	VAR jointtarget CDP_3887 := [[1.75, 35.13, 7.04, 0, 47.83, -268.25], [9E9, 9E9, 9E9, 9E9, 9E9, 9E9]];
	VAR jointtarget CDP_3888 := [[0.64, 35.11, 7.08, 0, 47.81, -269.36], [9E9, 9E9, 9E9, 9E9, 9E9, 9E9]];
	VAR jointtarget CDP_3889 := [[-0.47, 35.1, 7.09, 0, 47.81, -270.47], [9E9, 9E9, 9E9, 9E9, 9E9, 9E9]];
	VAR jointtarget CDP_3890 := [[-1.58, 35.13, 7.05, 0, 47.82, -271.58], [9E9, 9E9, 9E9, 9E9, 9E9, 9E9]];
	VAR jointtarget CDP_3891 := [[-2.69, 35.17, 6.97, 0, 47.86, -272.69], [9E9, 9E9, 9E9, 9E9, 9E9, 9E9]];
	VAR jointtarget CDP_3892 := [[-3.8, 35.24, 6.86, 0, 47.9, -273.8], [9E9, 9E9, 9E9, 9E9, 9E9, 9E9]];
	VAR jointtarget CDP_3893 := [[-4.9, 35.33, 6.71, 0, 47.97, -274.9], [9E9, 9E9, 9E9, 9E9, 9E9, 9E9]];
	VAR jointtarget CDP_3894 := [[-6, 35.44, 6.51, 0, 48.05, -276], [9E9, 9E9, 9E9, 9E9, 9E9, 9E9]];
	VAR jointtarget CDP_3895 := [[-7.1, 35.58, 6.28, 0, 48.14, -277.1], [9E9, 9E9, 9E9, 9E9, 9E9, 9E9]];
	VAR jointtarget CDP_3896 := [[-8.19, 35.73, 6.01, 0, 48.25, -278.19], [9E9, 9E9, 9E9, 9E9, 9E9, 9E9]];
	VAR jointtarget CDP_3897 := [[-9.28, 35.92, 5.7, 0, 48.38, -279.28], [9E9, 9E9, 9E9, 9E9, 9E9, 9E9]];
	VAR jointtarget CDP_3898 := [[-10.36, 36.12, 5.35, 0, 48.53, -280.36], [9E9, 9E9, 9E9, 9E9, 9E9, 9E9]];
	VAR jointtarget CDP_3899 := [[-11.43, 36.35, 4.96, 0, 48.69, -281.43], [9E9, 9E9, 9E9, 9E9, 9E9, 9E9]];
	VAR jointtarget CDP_3900 := [[-11.44, 36.35, 4.96, 0, 48.69, -281.78], [9E9, 9E9, 9E9, 9E9, 9E9, 9E9]];
	VAR jointtarget CDP_3901 := [[-11.46, 36.35, 4.95, 0, 48.7, -282.45], [9E9, 9E9, 9E9, 9E9, 9E9, 9E9]];
	VAR jointtarget CDP_3902 := [[-11.48, 36.36, 4.94, 0, 48.7, -283.13], [9E9, 9E9, 9E9, 9E9, 9E9, 9E9]];
	VAR jointtarget CDP_3903 := [[-11.49, 36.36, 4.94, 0, 48.7, -283.81], [9E9, 9E9, 9E9, 9E9, 9E9, 9E9]];
	VAR jointtarget CDP_3904 := [[-11.51, 36.37, 4.93, 0, 48.7, -284.49], [9E9, 9E9, 9E9, 9E9, 9E9, 9E9]];
	VAR jointtarget CDP_3905 := [[-11.53, 36.37, 4.92, 0, 48.71, -285.17], [9E9, 9E9, 9E9, 9E9, 9E9, 9E9]];
	VAR jointtarget CDP_3906 := [[-11.54, 36.38, 4.91, 0, 48.71, -285.84], [9E9, 9E9, 9E9, 9E9, 9E9, 9E9]];
	VAR jointtarget CDP_3907 := [[-11.56, 36.38, 4.9, 0, 48.72, -286.52], [9E9, 9E9, 9E9, 9E9, 9E9, 9E9]];
	VAR jointtarget CDP_3908 := [[-11.57, 36.39, 4.89, 0, 48.72, -287.2], [9E9, 9E9, 9E9, 9E9, 9E9, 9E9]];
	VAR jointtarget CDP_3909 := [[-11.59, 36.39, 4.88, 0, 48.72, -287.88], [9E9, 9E9, 9E9, 9E9, 9E9, 9E9]];
	VAR jointtarget CDP_3910 := [[-11.6, 36.4, 4.87, 0, 48.73, -288.56], [9E9, 9E9, 9E9, 9E9, 9E9, 9E9]];
	VAR jointtarget CDP_3911 := [[-11.62, 36.4, 4.86, 0, 48.73, -289.23], [9E9, 9E9, 9E9, 9E9, 9E9, 9E9]];
	VAR jointtarget CDP_3912 := [[-11.64, 36.41, 4.85, 0, 48.74, -289.91], [9E9, 9E9, 9E9, 9E9, 9E9, 9E9]];
	VAR jointtarget CDP_3913 := [[-11.65, 36.42, 4.84, 0, 48.74, -290.59], [9E9, 9E9, 9E9, 9E9, 9E9, 9E9]];
	VAR jointtarget CDP_3914 := [[-11.67, 36.42, 4.83, 0, 48.75, -291.27], [9E9, 9E9, 9E9, 9E9, 9E9, 9E9]];
	VAR jointtarget CDP_3915 := [[-11.68, 36.43, 4.82, 0, 48.75, -291.94], [9E9, 9E9, 9E9, 9E9, 9E9, 9E9]];
	VAR jointtarget CDP_3916 := [[-11.7, 36.44, 4.81, 0, 48.76, -292.62], [9E9, 9E9, 9E9, 9E9, 9E9, 9E9]];
	VAR jointtarget CDP_3917 := [[-11.71, 36.44, 4.79, 0, 48.76, -293.3], [9E9, 9E9, 9E9, 9E9, 9E9, 9E9]];
	VAR jointtarget CDP_3918 := [[-11.73, 36.45, 4.78, 0, 48.77, -293.98], [9E9, 9E9, 9E9, 9E9, 9E9, 9E9]];
	VAR jointtarget CDP_3919 := [[-11.74, 36.46, 4.77, 0, 48.77, -294.65], [9E9, 9E9, 9E9, 9E9, 9E9, 9E9]];
	VAR jointtarget CDP_3920 := [[-11.8, 36.49, 4.71, 0, 48.79, -295.04], [9E9, 9E9, 9E9, 9E9, 9E9, 9E9]];
	VAR jointtarget CDP_3921 := [[-11.86, 36.52, 4.66, 0, 48.82, -295.11], [9E9, 9E9, 9E9, 9E9, 9E9, 9E9]];
	VAR jointtarget CDP_3922 := [[-11.93, 36.55, 4.61, 0, 48.84, -295.17], [9E9, 9E9, 9E9, 9E9, 9E9, 9E9]];
	VAR jointtarget CDP_3923 := [[-11.99, 36.59, 4.55, 0, 48.86, -295.23], [9E9, 9E9, 9E9, 9E9, 9E9, 9E9]];
	VAR jointtarget CDP_3924 := [[-12.05, 36.62, 4.5, 0, 48.88, -295.29], [9E9, 9E9, 9E9, 9E9, 9E9, 9E9]];
	VAR jointtarget CDP_3925 := [[-12.11, 36.65, 4.44, 0, 48.91, -295.35], [9E9, 9E9, 9E9, 9E9, 9E9, 9E9]];
	VAR jointtarget CDP_3926 := [[-12.17, 36.68, 4.39, 0, 48.93, -295.41], [9E9, 9E9, 9E9, 9E9, 9E9, 9E9]];
	VAR jointtarget CDP_3927 := [[-12.23, 36.71, 4.34, 0, 48.95, -295.47], [9E9, 9E9, 9E9, 9E9, 9E9, 9E9]];
	VAR jointtarget CDP_3928 := [[-12.29, 36.74, 4.28, 0, 48.98, -295.53], [9E9, 9E9, 9E9, 9E9, 9E9, 9E9]];
	VAR jointtarget CDP_3929 := [[-12.35, 36.78, 4.23, 0, 49, -295.59], [9E9, 9E9, 9E9, 9E9, 9E9, 9E9]];
	VAR jointtarget CDP_3930 := [[-12.41, 36.81, 4.17, 0, 49.02, -295.65], [9E9, 9E9, 9E9, 9E9, 9E9, 9E9]];
	VAR jointtarget CDP_3931 := [[-12.47, 36.84, 4.12, 0, 49.04, -295.71], [9E9, 9E9, 9E9, 9E9, 9E9, 9E9]];
	VAR jointtarget CDP_3932 := [[-12.53, 36.87, 4.06, 0, 49.07, -295.77], [9E9, 9E9, 9E9, 9E9, 9E9, 9E9]];
	VAR jointtarget CDP_3933 := [[-12.59, 36.9, 4, 0, 49.09, -295.83], [9E9, 9E9, 9E9, 9E9, 9E9, 9E9]];
	VAR jointtarget CDP_3934 := [[-12.65, 36.94, 3.95, 0, 49.11, -295.89], [9E9, 9E9, 9E9, 9E9, 9E9, 9E9]];
	VAR jointtarget CDP_3935 := [[-12.71, 36.97, 3.89, 0, 49.14, -295.95], [9E9, 9E9, 9E9, 9E9, 9E9, 9E9]];
	VAR jointtarget CDP_3936 := [[-12.77, 37, 3.84, 0, 49.16, -296.01], [9E9, 9E9, 9E9, 9E9, 9E9, 9E9]];
	VAR jointtarget CDP_3937 := [[-12.83, 37.03, 3.78, 0, 49.18, -296.07], [9E9, 9E9, 9E9, 9E9, 9E9, 9E9]];
	VAR jointtarget CDP_3938 := [[-12.89, 37.07, 3.73, 0, 49.21, -296.13], [9E9, 9E9, 9E9, 9E9, 9E9, 9E9]];
	VAR jointtarget CDP_3939 := [[-12.95, 37.1, 3.67, 0, 49.23, -296.19], [9E9, 9E9, 9E9, 9E9, 9E9, 9E9]];
	VAR jointtarget CDP_3940 := [[-13.07, 37.15, 3.58, 0, 49.27, -291.14], [9E9, 9E9, 9E9, 9E9, 9E9, 9E9]];
	VAR jointtarget CDP_3941 := [[-13.19, 37.18, 3.53, 0, 49.29, -280.95], [9E9, 9E9, 9E9, 9E9, 9E9, 9E9]];
	VAR jointtarget CDP_3942 := [[-13.32, 37.18, 3.53, 0, 49.29, -270.75], [9E9, 9E9, 9E9, 9E9, 9E9, 9E9]];
	VAR jointtarget CDP_3943 := [[-13.45, 37.16, 3.57, 0, 49.27, -260.55], [9E9, 9E9, 9E9, 9E9, 9E9, 9E9]];
	VAR jointtarget CDP_3944 := [[-13.57, 37.11, 3.65, 0, 49.24, -250.35], [9E9, 9E9, 9E9, 9E9, 9E9, 9E9]];
	VAR jointtarget CDP_3945 := [[-13.68, 37.04, 3.78, 0, 49.19, -240.14], [9E9, 9E9, 9E9, 9E9, 9E9, 9E9]];
	VAR jointtarget CDP_3946 := [[-13.78, 36.94, 3.94, 0, 49.12, -229.91], [9E9, 9E9, 9E9, 9E9, 9E9, 9E9]];
	VAR jointtarget CDP_3947 := [[-13.86, 36.83, 4.13, 0, 49.04, -219.67], [9E9, 9E9, 9E9, 9E9, 9E9, 9E9]];
	VAR jointtarget CDP_3948 := [[-13.93, 36.71, 4.34, 0, 48.95, -209.41], [9E9, 9E9, 9E9, 9E9, 9E9, 9E9]];
	VAR jointtarget CDP_3949 := [[-13.97, 36.57, 4.58, 0, 48.85, -199.13], [9E9, 9E9, 9E9, 9E9, 9E9, 9E9]];
	VAR jointtarget CDP_3950 := [[-13.99, 36.43, 4.82, 0, 48.75, -188.83], [9E9, 9E9, 9E9, 9E9, 9E9, 9E9]];
	VAR jointtarget CDP_3951 := [[-13.98, 36.29, 5.07, 0, 48.65, -178.5], [9E9, 9E9, 9E9, 9E9, 9E9, 9E9]];
	VAR jointtarget CDP_3952 := [[-13.96, 36.14, 5.31, 0, 48.55, -168.15], [9E9, 9E9, 9E9, 9E9, 9E9, 9E9]];
	VAR jointtarget CDP_3953 := [[-13.91, 36.01, 5.54, 0, 48.45, -157.77], [9E9, 9E9, 9E9, 9E9, 9E9, 9E9]];
	VAR jointtarget CDP_3954 := [[-13.84, 35.89, 5.74, 0, 48.37, -147.38], [9E9, 9E9, 9E9, 9E9, 9E9, 9E9]];
	VAR jointtarget CDP_3955 := [[-13.75, 35.79, 5.92, 0, 48.29, -136.97], [9E9, 9E9, 9E9, 9E9, 9E9, 9E9]];
	VAR jointtarget CDP_3956 := [[-13.64, 35.7, 6.07, 0, 48.23, -126.54], [9E9, 9E9, 9E9, 9E9, 9E9, 9E9]];
	VAR jointtarget CDP_3957 := [[-13.52, 35.64, 6.17, 0, 48.19, -116.09], [9E9, 9E9, 9E9, 9E9, 9E9, 9E9]];
	VAR jointtarget CDP_3958 := [[-13.4, 35.6, 6.24, 0, 48.16, -105.64], [9E9, 9E9, 9E9, 9E9, 9E9, 9E9]];
	VAR jointtarget CDP_3959 := [[-13.27, 35.59, 6.26, 0, 48.15, -95.19], [9E9, 9E9, 9E9, 9E9, 9E9, 9E9]];
	VAR jointtarget CDP_3960 := [[-13.2, 35.59, 6.26, 0, 48.15, -89.96], [9E9, 9E9, 9E9, 9E9, 9E9, 9E9]];
	VAR jointtarget CDP_3961 := [[-13.13, 35.59, 6.26, 0, 48.15, -89.89], [9E9, 9E9, 9E9, 9E9, 9E9, 9E9]];
	VAR jointtarget CDP_3962 := [[-13.06, 35.59, 6.26, 0, 48.15, -89.82], [9E9, 9E9, 9E9, 9E9, 9E9, 9E9]];
	VAR jointtarget CDP_3963 := [[-12.99, 35.59, 6.26, 0, 48.15, -89.75], [9E9, 9E9, 9E9, 9E9, 9E9, 9E9]];
	VAR jointtarget CDP_3964 := [[-12.93, 35.59, 6.26, 0, 48.15, -89.69], [9E9, 9E9, 9E9, 9E9, 9E9, 9E9]];
	VAR jointtarget CDP_3965 := [[-12.86, 35.59, 6.26, 0, 48.16, -89.62], [9E9, 9E9, 9E9, 9E9, 9E9, 9E9]];
	VAR jointtarget CDP_3966 := [[-12.79, 35.59, 6.26, 0, 48.16, -89.55], [9E9, 9E9, 9E9, 9E9, 9E9, 9E9]];
	VAR jointtarget CDP_3967 := [[-12.72, 35.59, 6.26, 0, 48.16, -89.48], [9E9, 9E9, 9E9, 9E9, 9E9, 9E9]];
	VAR jointtarget CDP_3968 := [[-12.65, 35.59, 6.25, 0, 48.16, -89.41], [9E9, 9E9, 9E9, 9E9, 9E9, 9E9]];
	VAR jointtarget CDP_3969 := [[-12.59, 35.59, 6.25, 0, 48.16, -89.35], [9E9, 9E9, 9E9, 9E9, 9E9, 9E9]];
	VAR jointtarget CDP_3970 := [[-12.52, 35.59, 6.25, 0, 48.16, -89.28], [9E9, 9E9, 9E9, 9E9, 9E9, 9E9]];
	VAR jointtarget CDP_3971 := [[-12.45, 35.59, 6.25, 0, 48.16, -89.21], [9E9, 9E9, 9E9, 9E9, 9E9, 9E9]];
	VAR jointtarget CDP_3972 := [[-12.38, 35.59, 6.25, 0, 48.16, -89.14], [9E9, 9E9, 9E9, 9E9, 9E9, 9E9]];
	VAR jointtarget CDP_3973 := [[-12.32, 35.59, 6.25, 0, 48.17, -89.07], [9E9, 9E9, 9E9, 9E9, 9E9, 9E9]];
	VAR jointtarget CDP_3974 := [[-12.25, 35.59, 6.24, 0, 48.17, -89.01], [9E9, 9E9, 9E9, 9E9, 9E9, 9E9]];
	VAR jointtarget CDP_3975 := [[-12.18, 35.59, 6.24, 0, 48.17, -88.94], [9E9, 9E9, 9E9, 9E9, 9E9, 9E9]];
	VAR jointtarget CDP_3976 := [[-12.11, 35.59, 6.24, 0, 48.17, -88.87], [9E9, 9E9, 9E9, 9E9, 9E9, 9E9]];
	VAR jointtarget CDP_3977 := [[-12.04, 35.59, 6.24, 0, 48.17, -88.8], [9E9, 9E9, 9E9, 9E9, 9E9, 9E9]];
	VAR jointtarget CDP_3978 := [[-11.98, 35.59, 6.23, 0, 48.17, -88.74], [9E9, 9E9, 9E9, 9E9, 9E9, 9E9]];
	VAR jointtarget CDP_3979 := [[-11.91, 35.59, 6.23, 0, 48.18, -88.67], [9E9, 9E9, 9E9, 9E9, 9E9, 9E9]];
	VAR jointtarget CDP_3980 := [[-11.89, 35.59, 6.23, 0, 48.18, -88.98], [9E9, 9E9, 9E9, 9E9, 9E9, 9E9]];
	VAR jointtarget CDP_3981 := [[-11.87, 35.59, 6.23, 0, 48.18, -89.63], [9E9, 9E9, 9E9, 9E9, 9E9, 9E9]];
	VAR jointtarget CDP_3982 := [[-11.86, 35.59, 6.23, 0, 48.18, -90.27], [9E9, 9E9, 9E9, 9E9, 9E9, 9E9]];
	VAR jointtarget CDP_3983 := [[-11.84, 35.59, 6.23, 0, 48.18, -90.92], [9E9, 9E9, 9E9, 9E9, 9E9, 9E9]];
	VAR jointtarget CDP_3984 := [[-11.82, 35.59, 6.23, 0, 48.18, -91.56], [9E9, 9E9, 9E9, 9E9, 9E9, 9E9]];
	VAR jointtarget CDP_3985 := [[-11.81, 35.59, 6.23, 0, 48.18, -92.21], [9E9, 9E9, 9E9, 9E9, 9E9, 9E9]];
	VAR jointtarget CDP_3986 := [[-11.79, 35.59, 6.23, 0, 48.18, -92.85], [9E9, 9E9, 9E9, 9E9, 9E9, 9E9]];
	VAR jointtarget CDP_3987 := [[-11.77, 35.59, 6.24, 0, 48.18, -93.5], [9E9, 9E9, 9E9, 9E9, 9E9, 9E9]];
	VAR jointtarget CDP_3988 := [[-11.76, 35.59, 6.24, 0, 48.17, -94.14], [9E9, 9E9, 9E9, 9E9, 9E9, 9E9]];
	VAR jointtarget CDP_3989 := [[-11.74, 35.59, 6.24, 0, 48.17, -94.79], [9E9, 9E9, 9E9, 9E9, 9E9, 9E9]];
	VAR jointtarget CDP_3990 := [[-11.72, 35.58, 6.24, 0, 48.17, -95.43], [9E9, 9E9, 9E9, 9E9, 9E9, 9E9]];
	VAR jointtarget CDP_3991 := [[-11.71, 35.58, 6.25, 0, 48.17, -96.08], [9E9, 9E9, 9E9, 9E9, 9E9, 9E9]];
	VAR jointtarget CDP_3992 := [[-11.69, 35.58, 6.25, 0, 48.17, -96.72], [9E9, 9E9, 9E9, 9E9, 9E9, 9E9]];
	VAR jointtarget CDP_3993 := [[-11.67, 35.58, 6.25, 0, 48.17, -97.37], [9E9, 9E9, 9E9, 9E9, 9E9, 9E9]];
	VAR jointtarget CDP_3994 := [[-11.66, 35.57, 6.26, 0, 48.17, -98.01], [9E9, 9E9, 9E9, 9E9, 9E9, 9E9]];
	VAR jointtarget CDP_3995 := [[-11.64, 35.57, 6.26, 0, 48.16, -98.66], [9E9, 9E9, 9E9, 9E9, 9E9, 9E9]];
	VAR jointtarget CDP_3996 := [[-11.62, 35.57, 6.27, 0, 48.16, -99.31], [9E9, 9E9, 9E9, 9E9, 9E9, 9E9]];
	VAR jointtarget CDP_3997 := [[-11.61, 35.57, 6.27, 0, 48.16, -99.95], [9E9, 9E9, 9E9, 9E9, 9E9, 9E9]];
	VAR jointtarget CDP_3998 := [[-11.59, 35.56, 6.28, 0, 48.16, -100.6], [9E9, 9E9, 9E9, 9E9, 9E9, 9E9]];
	VAR jointtarget CDP_3999 := [[-11.57, 35.56, 6.29, 0, 48.16, -101.24], [9E9, 9E9, 9E9, 9E9, 9E9, 9E9]];
	VAR jointtarget CDP_4000 := [[-10.48, 35.33, 6.68, 0, 47.99, -100.48], [9E9, 9E9, 9E9, 9E9, 9E9, 9E9]];
	VAR jointtarget CDP_4001 := [[-9.38, 35.12, 7.03, 0, 47.85, -99.38], [9E9, 9E9, 9E9, 9E9, 9E9, 9E9]];
	VAR jointtarget CDP_4002 := [[-8.27, 34.94, 7.34, 0, 47.72, -98.27], [9E9, 9E9, 9E9, 9E9, 9E9, 9E9]];
	VAR jointtarget CDP_4003 := [[-7.15, 34.78, 7.61, 0, 47.61, -97.15], [9E9, 9E9, 9E9, 9E9, 9E9, 9E9]];
	VAR jointtarget CDP_4004 := [[-6.03, 34.64, 7.85, 0, 47.51, -96.03], [9E9, 9E9, 9E9, 9E9, 9E9, 9E9]];
	VAR jointtarget CDP_4005 := [[-4.9, 34.53, 8.04, 0, 47.43, -94.9], [9E9, 9E9, 9E9, 9E9, 9E9, 9E9]];
	VAR jointtarget CDP_4006 := [[-3.77, 34.44, 8.19, 0, 47.37, -93.77], [9E9, 9E9, 9E9, 9E9, 9E9, 9E9]];
	VAR jointtarget CDP_4007 := [[-2.64, 34.37, 8.31, 0, 47.32, -92.64], [9E9, 9E9, 9E9, 9E9, 9E9, 9E9]];
	VAR jointtarget CDP_4008 := [[-1.51, 34.33, 8.38, 0, 47.29, -91.51], [9E9, 9E9, 9E9, 9E9, 9E9, 9E9]];
	VAR jointtarget CDP_4009 := [[-0.37, 34.31, 8.41, 0, 47.28, -90.37], [9E9, 9E9, 9E9, 9E9, 9E9, 9E9]];
	VAR jointtarget CDP_4010 := [[0.76, 34.31, 8.41, 0, 47.28, -89.24], [9E9, 9E9, 9E9, 9E9, 9E9, 9E9]];
	VAR jointtarget CDP_4011 := [[1.9, 34.34, 8.36, 0, 47.3, -88.1], [9E9, 9E9, 9E9, 9E9, 9E9, 9E9]];
	VAR jointtarget CDP_4012 := [[3.03, 34.39, 8.27, 0, 47.34, -86.97], [9E9, 9E9, 9E9, 9E9, 9E9, 9E9]];
	VAR jointtarget CDP_4013 := [[4.16, 34.47, 8.14, 0, 47.39, -85.84], [9E9, 9E9, 9E9, 9E9, 9E9, 9E9]];
	VAR jointtarget CDP_4014 := [[5.29, 34.57, 7.98, 0, 47.46, -84.71], [9E9, 9E9, 9E9, 9E9, 9E9, 9E9]];
	VAR jointtarget CDP_4015 := [[6.42, 34.69, 7.77, 0, 47.54, -83.58], [9E9, 9E9, 9E9, 9E9, 9E9, 9E9]];
	VAR jointtarget CDP_4016 := [[7.54, 34.83, 7.52, 0, 47.64, -82.46], [9E9, 9E9, 9E9, 9E9, 9E9, 9E9]];
	VAR jointtarget CDP_4017 := [[8.65, 35, 7.24, 0, 47.76, -81.35], [9E9, 9E9, 9E9, 9E9, 9E9, 9E9]];
	VAR jointtarget CDP_4018 := [[9.76, 35.19, 6.91, 0, 47.9, -80.24], [9E9, 9E9, 9E9, 9E9, 9E9, 9E9]];
	VAR jointtarget CDP_4019 := [[10.86, 35.41, 6.55, 0, 48.05, -79.14], [9E9, 9E9, 9E9, 9E9, 9E9, 9E9]];
	VAR jointtarget CDP_4020 := [[10.87, 35.41, 6.54, 0, 48.05, -79.46], [9E9, 9E9, 9E9, 9E9, 9E9, 9E9]];
	VAR jointtarget CDP_4021 := [[10.89, 35.41, 6.54, 0, 48.05, -80.1], [9E9, 9E9, 9E9, 9E9, 9E9, 9E9]];
	VAR jointtarget CDP_4022 := [[10.91, 35.42, 6.53, 0, 48.05, -80.75], [9E9, 9E9, 9E9, 9E9, 9E9, 9E9]];
	VAR jointtarget CDP_4023 := [[10.92, 35.42, 6.53, 0, 48.06, -81.39], [9E9, 9E9, 9E9, 9E9, 9E9, 9E9]];
	VAR jointtarget CDP_4024 := [[10.94, 35.42, 6.52, 0, 48.06, -82.04], [9E9, 9E9, 9E9, 9E9, 9E9, 9E9]];
	VAR jointtarget CDP_4025 := [[10.96, 35.42, 6.52, 0, 48.06, -82.68], [9E9, 9E9, 9E9, 9E9, 9E9, 9E9]];
	VAR jointtarget CDP_4026 := [[10.97, 35.43, 6.51, 0, 48.06, -83.33], [9E9, 9E9, 9E9, 9E9, 9E9, 9E9]];
	VAR jointtarget CDP_4027 := [[10.99, 35.43, 6.51, 0, 48.06, -83.97], [9E9, 9E9, 9E9, 9E9, 9E9, 9E9]];
	VAR jointtarget CDP_4028 := [[11.01, 35.43, 6.51, 0, 48.06, -84.62], [9E9, 9E9, 9E9, 9E9, 9E9, 9E9]];
	VAR jointtarget CDP_4029 := [[11.02, 35.43, 6.51, 0, 48.06, -85.27], [9E9, 9E9, 9E9, 9E9, 9E9, 9E9]];
	VAR jointtarget CDP_4030 := [[11.04, 35.43, 6.5, 0, 48.07, -85.91], [9E9, 9E9, 9E9, 9E9, 9E9, 9E9]];
	VAR jointtarget CDP_4031 := [[11.06, 35.43, 6.5, 0, 48.07, -86.56], [9E9, 9E9, 9E9, 9E9, 9E9, 9E9]];
	VAR jointtarget CDP_4032 := [[11.07, 35.43, 6.5, 0, 48.07, -87.2], [9E9, 9E9, 9E9, 9E9, 9E9, 9E9]];
	VAR jointtarget CDP_4033 := [[11.09, 35.43, 6.5, 0, 48.07, -87.85], [9E9, 9E9, 9E9, 9E9, 9E9, 9E9]];
	VAR jointtarget CDP_4034 := [[11.11, 35.43, 6.5, 0, 48.07, -88.49], [9E9, 9E9, 9E9, 9E9, 9E9, 9E9]];
	VAR jointtarget CDP_4035 := [[11.13, 35.43, 6.5, 0, 48.07, -89.14], [9E9, 9E9, 9E9, 9E9, 9E9, 9E9]];
	VAR jointtarget CDP_4036 := [[11.14, 35.43, 6.5, 0, 48.07, -89.78], [9E9, 9E9, 9E9, 9E9, 9E9, 9E9]];
	VAR jointtarget CDP_4037 := [[11.16, 35.43, 6.5, 0, 48.07, -90.43], [9E9, 9E9, 9E9, 9E9, 9E9, 9E9]];
	VAR jointtarget CDP_4038 := [[11.18, 35.43, 6.5, 0, 48.07, -91.07], [9E9, 9E9, 9E9, 9E9, 9E9, 9E9]];
	VAR jointtarget CDP_4039 := [[11.19, 35.43, 6.5, 0, 48.07, -91.72], [9E9, 9E9, 9E9, 9E9, 9E9, 9E9]];
	VAR jointtarget CDP_4040 := [[11.26, 35.43, 6.5, 0, 48.07, -91.98], [9E9, 9E9, 9E9, 9E9, 9E9, 9E9]];
	VAR jointtarget CDP_4041 := [[11.33, 35.43, 6.51, 0, 48.06, -91.91], [9E9, 9E9, 9E9, 9E9, 9E9, 9E9]];
	VAR jointtarget CDP_4042 := [[11.4, 35.43, 6.51, 0, 48.06, -91.84], [9E9, 9E9, 9E9, 9E9, 9E9, 9E9]];
	VAR jointtarget CDP_4043 := [[11.47, 35.42, 6.52, 0, 48.06, -91.78], [9E9, 9E9, 9E9, 9E9, 9E9, 9E9]];
	VAR jointtarget CDP_4044 := [[11.53, 35.42, 6.52, 0, 48.06, -91.71], [9E9, 9E9, 9E9, 9E9, 9E9, 9E9]];
	VAR jointtarget CDP_4045 := [[11.6, 35.42, 6.52, 0, 48.06, -91.64], [9E9, 9E9, 9E9, 9E9, 9E9, 9E9]];
	VAR jointtarget CDP_4046 := [[11.67, 35.42, 6.53, 0, 48.06, -91.57], [9E9, 9E9, 9E9, 9E9, 9E9, 9E9]];
	VAR jointtarget CDP_4047 := [[11.74, 35.42, 6.53, 0, 48.05, -91.5], [9E9, 9E9, 9E9, 9E9, 9E9, 9E9]];
	VAR jointtarget CDP_4048 := [[11.81, 35.41, 6.53, 0, 48.05, -91.44], [9E9, 9E9, 9E9, 9E9, 9E9, 9E9]];
	VAR jointtarget CDP_4049 := [[11.87, 35.41, 6.54, 0, 48.05, -91.37], [9E9, 9E9, 9E9, 9E9, 9E9, 9E9]];
	VAR jointtarget CDP_4050 := [[11.94, 35.41, 6.54, 0, 48.05, -91.3], [9E9, 9E9, 9E9, 9E9, 9E9, 9E9]];
	VAR jointtarget CDP_4051 := [[12.01, 35.41, 6.54, 0, 48.05, -91.23], [9E9, 9E9, 9E9, 9E9, 9E9, 9E9]];
	VAR jointtarget CDP_4052 := [[12.08, 35.41, 6.54, 0, 48.05, -91.16], [9E9, 9E9, 9E9, 9E9, 9E9, 9E9]];
	VAR jointtarget CDP_4053 := [[12.15, 35.41, 6.55, 0, 48.05, -91.09], [9E9, 9E9, 9E9, 9E9, 9E9, 9E9]];
	VAR jointtarget CDP_4054 := [[12.21, 35.4, 6.55, 0, 48.05, -91.03], [9E9, 9E9, 9E9, 9E9, 9E9, 9E9]];
	VAR jointtarget CDP_4055 := [[12.28, 35.4, 6.55, 0, 48.05, -90.96], [9E9, 9E9, 9E9, 9E9, 9E9, 9E9]];
	VAR jointtarget CDP_4056 := [[12.35, 35.4, 6.55, 0, 48.04, -90.89], [9E9, 9E9, 9E9, 9E9, 9E9, 9E9]];
	VAR jointtarget CDP_4057 := [[12.42, 35.4, 6.56, 0, 48.04, -90.82], [9E9, 9E9, 9E9, 9E9, 9E9, 9E9]];
	VAR jointtarget CDP_4058 := [[12.49, 35.4, 6.56, 0, 48.04, -90.75], [9E9, 9E9, 9E9, 9E9, 9E9, 9E9]];
	VAR jointtarget CDP_4059 := [[12.55, 35.4, 6.56, 0, 48.04, -90.69], [9E9, 9E9, 9E9, 9E9, 9E9, 9E9]];
	VAR jointtarget CDP_4060 := [[12.69, 35.41, 6.54, 0, 48.05, -85.39], [9E9, 9E9, 9E9, 9E9, 9E9, 9E9]];
	VAR jointtarget CDP_4061 := [[12.81, 35.45, 6.48, 0, 48.08, -74.94], [9E9, 9E9, 9E9, 9E9, 9E9, 9E9]];
	VAR jointtarget CDP_4062 := [[12.93, 35.51, 6.37, 0, 48.12, -64.5], [9E9, 9E9, 9E9, 9E9, 9E9, 9E9]];
	VAR jointtarget CDP_4063 := [[13.04, 35.59, 6.23, 0, 48.18, -54.07], [9E9, 9E9, 9E9, 9E9, 9E9, 9E9]];
	VAR jointtarget CDP_4064 := [[13.13, 35.69, 6.05, 0, 48.25, -43.65], [9E9, 9E9, 9E9, 9E9, 9E9, 9E9]];
	VAR jointtarget CDP_4065 := [[13.2, 35.81, 5.85, 0, 48.34, -33.25], [9E9, 9E9, 9E9, 9E9, 9E9, 9E9]];
	VAR jointtarget CDP_4066 := [[13.25, 35.95, 5.62, 0, 48.43, -22.88], [9E9, 9E9, 9E9, 9E9, 9E9, 9E9]];
	VAR jointtarget CDP_4067 := [[13.28, 36.09, 5.39, 0, 48.53, -12.53], [9E9, 9E9, 9E9, 9E9, 9E9, 9E9]];
	VAR jointtarget CDP_4068 := [[13.29, 36.23, 5.14, 0, 48.63, -2.2], [9E9, 9E9, 9E9, 9E9, 9E9, 9E9]];
	VAR jointtarget CDP_4069 := [[13.27, 36.37, 4.9, 0, 48.73, 8.11], [9E9, 9E9, 9E9, 9E9, 9E9, 9E9]];
	VAR jointtarget CDP_4070 := [[13.23, 36.51, 4.66, 0, 48.83, 18.39], [9E9, 9E9, 9E9, 9E9, 9E9, 9E9]];
	VAR jointtarget CDP_4071 := [[13.17, 36.63, 4.45, 0, 48.92, 28.65], [9E9, 9E9, 9E9, 9E9, 9E9, 9E9]];
	VAR jointtarget CDP_4072 := [[13.08, 36.75, 4.25, 0, 49, 38.9], [9E9, 9E9, 9E9, 9E9, 9E9, 9E9]];
	VAR jointtarget CDP_4073 := [[12.99, 36.84, 4.09, 0, 49.07, 49.12], [9E9, 9E9, 9E9, 9E9, 9E9, 9E9]];
	VAR jointtarget CDP_4074 := [[12.88, 36.91, 3.97, 0, 49.12, 59.33], [9E9, 9E9, 9E9, 9E9, 9E9, 9E9]];
	VAR jointtarget CDP_4075 := [[12.75, 36.96, 3.88, 0, 49.16, 69.54], [9E9, 9E9, 9E9, 9E9, 9E9, 9E9]];
	VAR jointtarget CDP_4076 := [[12.63, 36.99, 3.83, 0, 49.18, 79.73], [9E9, 9E9, 9E9, 9E9, 9E9, 9E9]];
	VAR jointtarget CDP_4077 := [[12.5, 36.99, 3.83, 0, 49.18, 89.93], [9E9, 9E9, 9E9, 9E9, 9E9, 9E9]];
	VAR jointtarget CDP_4078 := [[12.37, 36.96, 3.88, 0, 49.16, 100.13], [9E9, 9E9, 9E9, 9E9, 9E9, 9E9]];
	VAR jointtarget CDP_4079 := [[12.25, 36.91, 3.97, 0, 49.12, 110.33], [9E9, 9E9, 9E9, 9E9, 9E9, 9E9]];
	VAR jointtarget CDP_4080 := [[12.19, 36.88, 4.02, 0, 49.1, 115.43], [9E9, 9E9, 9E9, 9E9, 9E9, 9E9]];
	VAR jointtarget CDP_4081 := [[12.13, 36.85, 4.07, 0, 49.08, 115.37], [9E9, 9E9, 9E9, 9E9, 9E9, 9E9]];
	VAR jointtarget CDP_4082 := [[12.07, 36.82, 4.13, 0, 49.05, 115.31], [9E9, 9E9, 9E9, 9E9, 9E9, 9E9]];
	VAR jointtarget CDP_4083 := [[12.01, 36.79, 4.18, 0, 49.03, 115.25], [9E9, 9E9, 9E9, 9E9, 9E9, 9E9]];
	VAR jointtarget CDP_4084 := [[11.95, 36.75, 4.24, 0, 49.01, 115.19], [9E9, 9E9, 9E9, 9E9, 9E9, 9E9]];
	VAR jointtarget CDP_4085 := [[11.89, 36.72, 4.29, 0, 48.99, 115.13], [9E9, 9E9, 9E9, 9E9, 9E9, 9E9]];
	VAR jointtarget CDP_4086 := [[11.83, 36.69, 4.35, 0, 48.96, 115.07], [9E9, 9E9, 9E9, 9E9, 9E9, 9E9]];
	VAR jointtarget CDP_4087 := [[11.77, 36.66, 4.4, 0, 48.94, 115.01], [9E9, 9E9, 9E9, 9E9, 9E9, 9E9]];
	VAR jointtarget CDP_4088 := [[11.71, 36.63, 4.45, 0, 48.92, 114.95], [9E9, 9E9, 9E9, 9E9, 9E9, 9E9]];
	VAR jointtarget CDP_4089 := [[11.65, 36.6, 4.51, 0, 48.9, 114.89], [9E9, 9E9, 9E9, 9E9, 9E9, 9E9]];
	VAR jointtarget CDP_4090 := [[11.59, 36.57, 4.56, 0, 48.87, 114.83], [9E9, 9E9, 9E9, 9E9, 9E9, 9E9]];
	VAR jointtarget CDP_4091 := [[11.53, 36.54, 4.61, 0, 48.85, 114.77], [9E9, 9E9, 9E9, 9E9, 9E9, 9E9]];
	VAR jointtarget CDP_4092 := [[11.47, 36.5, 4.67, 0, 48.83, 114.71], [9E9, 9E9, 9E9, 9E9, 9E9, 9E9]];
	VAR jointtarget CDP_4093 := [[11.4, 36.47, 4.72, 0, 48.81, 114.64], [9E9, 9E9, 9E9, 9E9, 9E9, 9E9]];
	VAR jointtarget CDP_4094 := [[11.34, 36.44, 4.77, 0, 48.78, 114.58], [9E9, 9E9, 9E9, 9E9, 9E9, 9E9]];
	VAR jointtarget CDP_4095 := [[11.28, 36.41, 4.83, 0, 48.76, 114.52], [9E9, 9E9, 9E9, 9E9, 9E9, 9E9]];
	VAR jointtarget CDP_4096 := [[11.22, 36.38, 4.88, 0, 48.74, 114.46], [9E9, 9E9, 9E9, 9E9, 9E9, 9E9]];
	VAR jointtarget CDP_4097 := [[11.16, 36.35, 4.93, 0, 48.72, 114.4], [9E9, 9E9, 9E9, 9E9, 9E9, 9E9]];
	VAR jointtarget CDP_4098 := [[11.1, 36.32, 4.98, 0, 48.7, 114.34], [9E9, 9E9, 9E9, 9E9, 9E9, 9E9]];
	VAR jointtarget CDP_4099 := [[11.04, 36.29, 5.03, 0, 48.68, 114.28], [9E9, 9E9, 9E9, 9E9, 9E9, 9E9]];
	VAR jointtarget CDP_4100 := [[11.02, 36.28, 5.05, 0, 48.67, 113.93], [9E9, 9E9, 9E9, 9E9, 9E9, 9E9]];
	VAR jointtarget CDP_4101 := [[11.01, 36.28, 5.06, 0, 48.66, 113.26], [9E9, 9E9, 9E9, 9E9, 9E9, 9E9]];
	VAR jointtarget CDP_4102 := [[10.99, 36.27, 5.07, 0, 48.66, 112.58], [9E9, 9E9, 9E9, 9E9, 9E9, 9E9]];
	VAR jointtarget CDP_4103 := [[10.98, 36.26, 5.08, 0, 48.65, 111.9], [9E9, 9E9, 9E9, 9E9, 9E9, 9E9]];
	VAR jointtarget CDP_4104 := [[10.96, 36.26, 5.09, 0, 48.65, 111.22], [9E9, 9E9, 9E9, 9E9, 9E9, 9E9]];
	VAR jointtarget CDP_4105 := [[10.95, 36.25, 5.11, 0, 48.65, 110.55], [9E9, 9E9, 9E9, 9E9, 9E9, 9E9]];
	VAR jointtarget CDP_4106 := [[10.93, 36.24, 5.12, 0, 48.64, 109.87], [9E9, 9E9, 9E9, 9E9, 9E9, 9E9]];
	VAR jointtarget CDP_4107 := [[10.91, 36.24, 5.13, 0, 48.64, 109.19], [9E9, 9E9, 9E9, 9E9, 9E9, 9E9]];
	VAR jointtarget CDP_4108 := [[10.9, 36.23, 5.14, 0, 48.63, 108.51], [9E9, 9E9, 9E9, 9E9, 9E9, 9E9]];
	VAR jointtarget CDP_4109 := [[10.88, 36.23, 5.15, 0, 48.63, 107.83], [9E9, 9E9, 9E9, 9E9, 9E9, 9E9]];
	VAR jointtarget CDP_4110 := [[10.87, 36.22, 5.16, 0, 48.62, 107.16], [9E9, 9E9, 9E9, 9E9, 9E9, 9E9]];
	VAR jointtarget CDP_4111 := [[10.85, 36.21, 5.16, 0, 48.62, 106.48], [9E9, 9E9, 9E9, 9E9, 9E9, 9E9]];
	VAR jointtarget CDP_4112 := [[10.83, 36.21, 5.17, 0, 48.62, 105.8], [9E9, 9E9, 9E9, 9E9, 9E9, 9E9]];
	VAR jointtarget CDP_4113 := [[10.82, 36.2, 5.18, 0, 48.61, 105.12], [9E9, 9E9, 9E9, 9E9, 9E9, 9E9]];
	VAR jointtarget CDP_4114 := [[10.8, 36.2, 5.19, 0, 48.61, 104.44], [9E9, 9E9, 9E9, 9E9, 9E9, 9E9]];
	VAR jointtarget CDP_4115 := [[10.79, 36.2, 5.2, 0, 48.61, 103.77], [9E9, 9E9, 9E9, 9E9, 9E9, 9E9]];
	VAR jointtarget CDP_4116 := [[10.77, 36.19, 5.2, 0, 48.6, 103.09], [9E9, 9E9, 9E9, 9E9, 9E9, 9E9]];
	VAR jointtarget CDP_4117 := [[10.75, 36.19, 5.21, 0, 48.6, 102.41], [9E9, 9E9, 9E9, 9E9, 9E9, 9E9]];
	VAR jointtarget CDP_4118 := [[10.74, 36.18, 5.22, 0, 48.6, 101.73], [9E9, 9E9, 9E9, 9E9, 9E9, 9E9]];
	VAR jointtarget CDP_4119 := [[10.72, 36.18, 5.22, 0, 48.6, 101.05], [9E9, 9E9, 9E9, 9E9, 9E9, 9E9]];
	VAR jointtarget CDP_4120 := [[9.64, 35.97, 5.58, 0, 48.45, 99.64], [9E9, 9E9, 9E9, 9E9, 9E9, 9E9]];
	VAR jointtarget CDP_4121 := [[8.56, 35.78, 5.91, 0, 48.31, 98.56], [9E9, 9E9, 9E9, 9E9, 9E9, 9E9]];
	VAR jointtarget CDP_4122 := [[7.47, 35.61, 6.19, 0, 48.19, 97.47], [9E9, 9E9, 9E9, 9E9, 9E9, 9E9]];
	VAR jointtarget CDP_4123 := [[6.38, 35.47, 6.44, 0, 48.09, 96.38], [9E9, 9E9, 9E9, 9E9, 9E9, 9E9]];
	VAR jointtarget CDP_4124 := [[5.28, 35.35, 6.64, 0, 48.01, 95.28], [9E9, 9E9, 9E9, 9E9, 9E9, 9E9]];
	VAR jointtarget CDP_4125 := [[4.17, 35.25, 6.81, 0, 47.94, 94.17], [9E9, 9E9, 9E9, 9E9, 9E9, 9E9]];
	VAR jointtarget CDP_4126 := [[3.07, 35.18, 6.94, 0, 47.89, 93.07], [9E9, 9E9, 9E9, 9E9, 9E9, 9E9]];
	VAR jointtarget CDP_4127 := [[1.96, 35.13, 7.03, 0, 47.85, 91.96], [9E9, 9E9, 9E9, 9E9, 9E9, 9E9]];
	VAR jointtarget CDP_4128 := [[0.85, 35.1, 7.07, 0, 47.83, 90.85], [9E9, 9E9, 9E9, 9E9, 9E9, 9E9]];
	VAR jointtarget CDP_4129 := [[-0.26, 35.09, 7.09, 0, 47.82, 89.74], [9E9, 9E9, 9E9, 9E9, 9E9, 9E9]];
	VAR jointtarget CDP_4130 := [[-1.37, 35.11, 7.06, 0, 47.84, 88.63], [9E9, 9E9, 9E9, 9E9, 9E9, 9E9]];
	VAR jointtarget CDP_4131 := [[-2.48, 35.15, 6.99, 0, 47.86, 87.52], [9E9, 9E9, 9E9, 9E9, 9E9, 9E9]];
	VAR jointtarget CDP_4132 := [[-3.59, 35.21, 6.88, 0, 47.91, 86.41], [9E9, 9E9, 9E9, 9E9, 9E9, 9E9]];
	VAR jointtarget CDP_4133 := [[-4.7, 35.3, 6.73, 0, 47.97, 85.3], [9E9, 9E9, 9E9, 9E9, 9E9, 9E9]];
	VAR jointtarget CDP_4134 := [[-5.8, 35.4, 6.55, 0, 48.05, 84.2], [9E9, 9E9, 9E9, 9E9, 9E9, 9E9]];
	VAR jointtarget CDP_4135 := [[-6.9, 35.54, 6.32, 0, 48.14, 83.1], [9E9, 9E9, 9E9, 9E9, 9E9, 9E9]];
	VAR jointtarget CDP_4136 := [[-7.99, 35.69, 6.06, 0, 48.25, 82.01], [9E9, 9E9, 9E9, 9E9, 9E9, 9E9]];
	VAR jointtarget CDP_4137 := [[-9.08, 35.87, 5.76, 0, 48.37, 80.92], [9E9, 9E9, 9E9, 9E9, 9E9, 9E9]];
	VAR jointtarget CDP_4138 := [[-10.16, 36.07, 5.42, 0, 48.52, 79.84], [9E9, 9E9, 9E9, 9E9, 9E9, 9E9]];
	VAR jointtarget CDP_4139 := [[-11.23, 36.29, 5.04, 0, 48.67, 78.77], [9E9, 9E9, 9E9, 9E9, 9E9, 9E9]];
	VAR jointtarget CDP_4140 := [[-11.28, 36.3, 5.02, 0, 48.68, 79.81], [9E9, 9E9, 9E9, 9E9, 9E9, 9E9]];
	VAR jointtarget CDP_4141 := [[-11.34, 36.31, 5, 0, 48.69, 81.95], [9E9, 9E9, 9E9, 9E9, 9E9, 9E9]];
	VAR jointtarget CDP_4142 := [[-11.39, 36.31, 4.99, 0, 48.69, 84.09], [9E9, 9E9, 9E9, 9E9, 9E9, 9E9]];
	VAR jointtarget CDP_4143 := [[-11.45, 36.32, 4.99, 0, 48.7, 86.23], [9E9, 9E9, 9E9, 9E9, 9E9, 9E9]];
	VAR jointtarget CDP_4144 := [[-11.5, 36.32, 4.98, 0, 48.7, 88.37], [9E9, 9E9, 9E9, 9E9, 9E9, 9E9]];
	VAR jointtarget CDP_4145 := [[-11.56, 36.32, 4.98, 0, 48.7, 90.51], [9E9, 9E9, 9E9, 9E9, 9E9, 9E9]];
	VAR jointtarget CDP_4146 := [[-11.61, 36.32, 4.99, 0, 48.69, 92.65], [9E9, 9E9, 9E9, 9E9, 9E9, 9E9]];
	VAR jointtarget CDP_4147 := [[-11.67, 36.31, 5, 0, 48.69, 94.78], [9E9, 9E9, 9E9, 9E9, 9E9, 9E9]];
	VAR jointtarget CDP_4148 := [[-11.72, 36.3, 5.01, 0, 48.69, 96.92], [9E9, 9E9, 9E9, 9E9, 9E9, 9E9]];
	VAR jointtarget CDP_4149 := [[-11.78, 36.29, 5.03, 0, 48.68, 99.06], [9E9, 9E9, 9E9, 9E9, 9E9, 9E9]];
	VAR jointtarget CDP_4150 := [[-11.83, 36.28, 5.05, 0, 48.67, 101.2], [9E9, 9E9, 9E9, 9E9, 9E9, 9E9]];
	VAR jointtarget CDP_4151 := [[-11.89, 36.27, 5.07, 0, 48.66, 103.34], [9E9, 9E9, 9E9, 9E9, 9E9, 9E9]];
	VAR jointtarget CDP_4152 := [[-11.94, 36.25, 5.1, 0, 48.65, 105.48], [9E9, 9E9, 9E9, 9E9, 9E9, 9E9]];
	VAR jointtarget CDP_4153 := [[-11.99, 36.23, 5.13, 0, 48.64, 107.63], [9E9, 9E9, 9E9, 9E9, 9E9, 9E9]];
	VAR jointtarget CDP_4154 := [[-12.04, 36.21, 5.17, 0, 48.62, 109.77], [9E9, 9E9, 9E9, 9E9, 9E9, 9E9]];
	VAR jointtarget CDP_4155 := [[-12.09, 36.19, 5.2, 0, 48.6, 111.91], [9E9, 9E9, 9E9, 9E9, 9E9, 9E9]];
	VAR jointtarget CDP_4156 := [[-12.15, 36.17, 5.25, 0, 48.59, 114.05], [9E9, 9E9, 9E9, 9E9, 9E9, 9E9]];
	VAR jointtarget CDP_4157 := [[-12.19, 36.14, 5.29, 0, 48.57, 116.2], [9E9, 9E9, 9E9, 9E9, 9E9, 9E9]];
	VAR jointtarget CDP_4158 := [[-12.24, 36.11, 5.34, 0, 48.55, 118.34], [9E9, 9E9, 9E9, 9E9, 9E9, 9E9]];
	VAR jointtarget CDP_4159 := [[-12.29, 36.08, 5.4, 0, 48.53, 120.49], [9E9, 9E9, 9E9, 9E9, 9E9, 9E9]];
	VAR jointtarget CDP_4160 := [[-12.32, 36.06, 5.43, 0, 48.51, 121.56], [9E9, 9E9, 9E9, 9E9, 9E9, 9E9]];
	VAR jointtarget CDP_4161 := [[-12.35, 36.04, 5.46, 0, 48.5, 121.53], [9E9, 9E9, 9E9, 9E9, 9E9, 9E9]];
	VAR jointtarget CDP_4162 := [[-12.38, 36.02, 5.49, 0, 48.48, 121.5], [9E9, 9E9, 9E9, 9E9, 9E9, 9E9]];
	VAR jointtarget CDP_4163 := [[-12.41, 36, 5.53, 0, 48.47, 121.47], [9E9, 9E9, 9E9, 9E9, 9E9, 9E9]];
	VAR jointtarget CDP_4164 := [[-12.43, 35.98, 5.56, 0, 48.46, 121.44], [9E9, 9E9, 9E9, 9E9, 9E9, 9E9]];
	VAR jointtarget CDP_4165 := [[-12.46, 35.97, 5.59, 0, 48.44, 121.41], [9E9, 9E9, 9E9, 9E9, 9E9, 9E9]];
	VAR jointtarget CDP_4166 := [[-12.49, 35.95, 5.62, 0, 48.43, 121.39], [9E9, 9E9, 9E9, 9E9, 9E9, 9E9]];
	VAR jointtarget CDP_4167 := [[-12.52, 35.93, 5.66, 0, 48.42, 121.36], [9E9, 9E9, 9E9, 9E9, 9E9, 9E9]];
	VAR jointtarget CDP_4168 := [[-12.55, 35.91, 5.69, 0, 48.4, 121.33], [9E9, 9E9, 9E9, 9E9, 9E9, 9E9]];
	VAR jointtarget CDP_4169 := [[-12.58, 35.89, 5.72, 0, 48.39, 121.3], [9E9, 9E9, 9E9, 9E9, 9E9, 9E9]];
	VAR jointtarget CDP_4170 := [[-12.61, 35.87, 5.75, 0, 48.38, 121.27], [9E9, 9E9, 9E9, 9E9, 9E9, 9E9]];
	VAR jointtarget CDP_4171 := [[-12.63, 35.85, 5.79, 0, 48.36, 121.24], [9E9, 9E9, 9E9, 9E9, 9E9, 9E9]];
	VAR jointtarget CDP_4172 := [[-12.66, 35.83, 5.82, 0, 48.35, 121.21], [9E9, 9E9, 9E9, 9E9, 9E9, 9E9]];
	VAR jointtarget CDP_4173 := [[-12.69, 35.81, 5.85, 0, 48.34, 121.18], [9E9, 9E9, 9E9, 9E9, 9E9, 9E9]];
	VAR jointtarget CDP_4174 := [[-12.72, 35.79, 5.88, 0, 48.32, 121.16], [9E9, 9E9, 9E9, 9E9, 9E9, 9E9]];
	VAR jointtarget CDP_4175 := [[-12.75, 35.78, 5.92, 0, 48.31, 121.13], [9E9, 9E9, 9E9, 9E9, 9E9, 9E9]];
	VAR jointtarget CDP_4176 := [[-12.78, 35.76, 5.95, 0, 48.3, 121.1], [9E9, 9E9, 9E9, 9E9, 9E9, 9E9]];
	VAR jointtarget CDP_4177 := [[-12.81, 35.74, 5.98, 0, 48.28, 121.07], [9E9, 9E9, 9E9, 9E9, 9E9, 9E9]];
	VAR jointtarget CDP_4178 := [[-12.84, 35.72, 6.01, 0, 48.27, 121.04], [9E9, 9E9, 9E9, 9E9, 9E9, 9E9]];
	VAR jointtarget CDP_4179 := [[-12.86, 35.7, 6.04, 0, 48.26, 121.01], [9E9, 9E9, 9E9, 9E9, 9E9, 9E9]];
	VAR jointtarget CDP_4180 := [[-13.02, 35.63, 6.17, 0, 48.2, 114.17], [9E9, 9E9, 9E9, 9E9, 9E9, 9E9]];
	VAR jointtarget CDP_4181 := [[-13.18, 35.59, 6.23, 0, 48.18, 100.62], [9E9, 9E9, 9E9, 9E9, 9E9, 9E9]];
	VAR jointtarget CDP_4182 := [[-13.34, 35.6, 6.21, 0, 48.19, 87.07], [9E9, 9E9, 9E9, 9E9, 9E9, 9E9]];
	VAR jointtarget CDP_4183 := [[-13.5, 35.65, 6.12, 0, 48.22, 73.52], [9E9, 9E9, 9E9, 9E9, 9E9, 9E9]];
	VAR jointtarget CDP_4184 := [[-13.64, 35.74, 5.97, 0, 48.29, 59.99], [9E9, 9E9, 9E9, 9E9, 9E9, 9E9]];
	VAR jointtarget CDP_4185 := [[-13.76, 35.87, 5.76, 0, 48.37, 46.48], [9E9, 9E9, 9E9, 9E9, 9E9, 9E9]];
	VAR jointtarget CDP_4186 := [[-13.85, 36.01, 5.51, 0, 48.48, 33.01], [9E9, 9E9, 9E9, 9E9, 9E9, 9E9]];
	VAR jointtarget CDP_4187 := [[-13.91, 36.18, 5.22, 0, 48.6, 19.56], [9E9, 9E9, 9E9, 9E9, 9E9, 9E9]];
	VAR jointtarget CDP_4188 := [[-13.92, 36.36, 4.91, 0, 48.73, 6.16], [9E9, 9E9, 9E9, 9E9, 9E9, 9E9]];
	VAR jointtarget CDP_4189 := [[-13.9, 36.54, 4.61, 0, 48.85, -7.21], [9E9, 9E9, 9E9, 9E9, 9E9, 9E9]];
	VAR jointtarget CDP_4190 := [[-13.85, 36.71, 4.32, 0, 48.97, -20.54], [9E9, 9E9, 9E9, 9E9, 9E9, 9E9]];
	VAR jointtarget CDP_4191 := [[-13.76, 36.86, 4.06, 0, 49.08, -33.84], [9E9, 9E9, 9E9, 9E9, 9E9, 9E9]];
	VAR jointtarget CDP_4192 := [[-13.64, 36.98, 3.85, 0, 49.17, -47.11], [9E9, 9E9, 9E9, 9E9, 9E9, 9E9]];
	VAR jointtarget CDP_4193 := [[-13.5, 37.07, 3.7, 0, 49.23, -60.35], [9E9, 9E9, 9E9, 9E9, 9E9, 9E9]];
	VAR jointtarget CDP_4194 := [[-13.34, 37.12, 3.61, 0, 49.27, -73.59], [9E9, 9E9, 9E9, 9E9, 9E9, 9E9]];
	VAR jointtarget CDP_4195 := [[-13.18, 37.13, 3.59, 0, 49.28, -86.81], [9E9, 9E9, 9E9, 9E9, 9E9, 9E9]];
	VAR jointtarget CDP_4196 := [[-13.02, 37.1, 3.65, 0, 49.26, -100.04], [9E9, 9E9, 9E9, 9E9, 9E9, 9E9]];
	VAR jointtarget CDP_4197 := [[-12.88, 37.03, 3.77, 0, 49.2, -113.28], [9E9, 9E9, 9E9, 9E9, 9E9, 9E9]];
	VAR jointtarget CDP_4198 := [[-12.75, 36.92, 3.96, 0, 49.13, -126.54], [9E9, 9E9, 9E9, 9E9, 9E9, 9E9]];
	VAR jointtarget CDP_4199 := [[-12.64, 36.78, 4.19, 0, 49.03, -139.82], [9E9, 9E9, 9E9, 9E9, 9E9, 9E9]];
	VAR jointtarget CDP_4200 := [[-12.62, 36.74, 4.26, 0, 49, -146.49], [9E9, 9E9, 9E9, 9E9, 9E9, 9E9]];
	VAR jointtarget CDP_4201 := [[-12.59, 36.7, 4.33, 0, 48.97, -146.47], [9E9, 9E9, 9E9, 9E9, 9E9, 9E9]];
	VAR jointtarget CDP_4202 := [[-12.57, 36.66, 4.4, 0, 48.94, -146.44], [9E9, 9E9, 9E9, 9E9, 9E9, 9E9]];
	VAR jointtarget CDP_4203 := [[-12.54, 36.62, 4.48, 0, 48.91, -146.42], [9E9, 9E9, 9E9, 9E9, 9E9, 9E9]];
	VAR jointtarget CDP_4204 := [[-12.52, 36.57, 4.55, 0, 48.88, -146.4], [9E9, 9E9, 9E9, 9E9, 9E9, 9E9]];
	VAR jointtarget CDP_4205 := [[-12.49, 36.53, 4.62, 0, 48.85, -146.37], [9E9, 9E9, 9E9, 9E9, 9E9, 9E9]];
	VAR jointtarget CDP_4206 := [[-12.47, 36.49, 4.69, 0, 48.82, -146.35], [9E9, 9E9, 9E9, 9E9, 9E9, 9E9]];
	VAR jointtarget CDP_4207 := [[-12.44, 36.45, 4.76, 0, 48.79, -146.32], [9E9, 9E9, 9E9, 9E9, 9E9, 9E9]];
	VAR jointtarget CDP_4208 := [[-12.42, 36.41, 4.83, 0, 48.76, -146.3], [9E9, 9E9, 9E9, 9E9, 9E9, 9E9]];
	VAR jointtarget CDP_4209 := [[-12.39, 36.37, 4.9, 0, 48.73, -146.27], [9E9, 9E9, 9E9, 9E9, 9E9, 9E9]];
	VAR jointtarget CDP_4210 := [[-12.37, 36.33, 4.97, 0, 48.7, -146.25], [9E9, 9E9, 9E9, 9E9, 9E9, 9E9]];
	VAR jointtarget CDP_4211 := [[-12.34, 36.29, 5.04, 0, 48.67, -146.22], [9E9, 9E9, 9E9, 9E9, 9E9, 9E9]];
	VAR jointtarget CDP_4212 := [[-12.32, 36.25, 5.11, 0, 48.64, -146.2], [9E9, 9E9, 9E9, 9E9, 9E9, 9E9]];
	VAR jointtarget CDP_4213 := [[-12.29, 36.2, 5.18, 0, 48.61, -146.17], [9E9, 9E9, 9E9, 9E9, 9E9, 9E9]];
	VAR jointtarget CDP_4214 := [[-12.27, 36.16, 5.25, 0, 48.58, -146.15], [9E9, 9E9, 9E9, 9E9, 9E9, 9E9]];
	VAR jointtarget CDP_4215 := [[-12.24, 36.12, 5.32, 0, 48.56, -146.12], [9E9, 9E9, 9E9, 9E9, 9E9, 9E9]];
	VAR jointtarget CDP_4216 := [[-12.22, 36.08, 5.39, 0, 48.53, -146.1], [9E9, 9E9, 9E9, 9E9, 9E9, 9E9]];
	VAR jointtarget CDP_4217 := [[-12.19, 36.04, 5.46, 0, 48.5, -146.07], [9E9, 9E9, 9E9, 9E9, 9E9, 9E9]];
	VAR jointtarget CDP_4218 := [[-12.17, 36, 5.53, 0, 48.47, -146.05], [9E9, 9E9, 9E9, 9E9, 9E9, 9E9]];
	VAR jointtarget CDP_4219 := [[-12.14, 35.96, 5.6, 0, 48.44, -146.02], [9E9, 9E9, 9E9, 9E9, 9E9, 9E9]];
	VAR jointtarget CDP_4220 := [[-12.14, 35.95, 5.62, 0, 48.43, -145.46], [9E9, 9E9, 9E9, 9E9, 9E9, 9E9]];
	VAR jointtarget CDP_4221 := [[-12.13, 35.93, 5.64, 0, 48.42, -144.35], [9E9, 9E9, 9E9, 9E9, 9E9, 9E9]];
	VAR jointtarget CDP_4222 := [[-12.12, 35.92, 5.66, 0, 48.41, -143.24], [9E9, 9E9, 9E9, 9E9, 9E9, 9E9]];
	VAR jointtarget CDP_4223 := [[-12.11, 35.91, 5.69, 0, 48.4, -142.13], [9E9, 9E9, 9E9, 9E9, 9E9, 9E9]];
	VAR jointtarget CDP_4224 := [[-12.1, 35.9, 5.71, 0, 48.4, -141.01], [9E9, 9E9, 9E9, 9E9, 9E9, 9E9]];
	VAR jointtarget CDP_4225 := [[-12.09, 35.89, 5.73, 0, 48.39, -139.9], [9E9, 9E9, 9E9, 9E9, 9E9, 9E9]];
	VAR jointtarget CDP_4226 := [[-12.08, 35.87, 5.75, 0, 48.38, -138.79], [9E9, 9E9, 9E9, 9E9, 9E9, 9E9]];
	VAR jointtarget CDP_4227 := [[-12.07, 35.86, 5.76, 0, 48.37, -137.68], [9E9, 9E9, 9E9, 9E9, 9E9, 9E9]];
	VAR jointtarget CDP_4228 := [[-12.06, 35.85, 5.78, 0, 48.36, -136.56], [9E9, 9E9, 9E9, 9E9, 9E9, 9E9]];
	VAR jointtarget CDP_4229 := [[-12.05, 35.84, 5.8, 0, 48.36, -135.45], [9E9, 9E9, 9E9, 9E9, 9E9, 9E9]];
	VAR jointtarget CDP_4230 := [[-12.04, 35.83, 5.82, 0, 48.35, -134.34], [9E9, 9E9, 9E9, 9E9, 9E9, 9E9]];
	VAR jointtarget CDP_4231 := [[-12.03, 35.82, 5.84, 0, 48.34, -133.22], [9E9, 9E9, 9E9, 9E9, 9E9, 9E9]];
	VAR jointtarget CDP_4232 := [[-12.02, 35.81, 5.86, 0, 48.34, -132.11], [9E9, 9E9, 9E9, 9E9, 9E9, 9E9]];
	VAR jointtarget CDP_4233 := [[-12.01, 35.8, 5.87, 0, 48.33, -130.99], [9E9, 9E9, 9E9, 9E9, 9E9, 9E9]];
	VAR jointtarget CDP_4234 := [[-12, 35.79, 5.89, 0, 48.32, -129.88], [9E9, 9E9, 9E9, 9E9, 9E9, 9E9]];
	VAR jointtarget CDP_4235 := [[-11.99, 35.78, 5.91, 0, 48.32, -128.76], [9E9, 9E9, 9E9, 9E9, 9E9, 9E9]];
	VAR jointtarget CDP_4236 := [[-11.98, 35.77, 5.92, 0, 48.31, -127.65], [9E9, 9E9, 9E9, 9E9, 9E9, 9E9]];
	VAR jointtarget CDP_4237 := [[-11.97, 35.76, 5.94, 0, 48.3, -126.53], [9E9, 9E9, 9E9, 9E9, 9E9, 9E9]];
	VAR jointtarget CDP_4238 := [[-11.96, 35.75, 5.95, 0, 48.3, -125.42], [9E9, 9E9, 9E9, 9E9, 9E9, 9E9]];
	VAR jointtarget CDP_4239 := [[-11.95, 35.74, 5.97, 0, 48.29, -124.3], [9E9, 9E9, 9E9, 9E9, 9E9, 9E9]];
	VAR jointtarget CDP_4240 := [[-11.94, 35.73, 5.98, 0, 48.29, -123.74], [9E9, 9E9, 9E9, 9E9, 9E9, 9E9]];
	VAR jointtarget CDP_4241 := [[-11.93, 35.72, 5.99, 0, 48.28, -123.73], [9E9, 9E9, 9E9, 9E9, 9E9, 9E9]];
	VAR jointtarget CDP_4242 := [[-11.92, 35.72, 6, 0, 48.28, -123.72], [9E9, 9E9, 9E9, 9E9, 9E9, 9E9]];
	VAR jointtarget CDP_4243 := [[-11.9, 35.71, 6.02, 0, 48.27, -123.71], [9E9, 9E9, 9E9, 9E9, 9E9, 9E9]];
	VAR jointtarget CDP_4244 := [[-11.89, 35.7, 6.03, 0, 48.27, -123.7], [9E9, 9E9, 9E9, 9E9, 9E9, 9E9]];
	VAR jointtarget CDP_4245 := [[-11.88, 35.69, 6.04, 0, 48.26, -123.69], [9E9, 9E9, 9E9, 9E9, 9E9, 9E9]];
	VAR jointtarget CDP_4246 := [[-11.87, 35.69, 6.06, 0, 48.26, -123.68], [9E9, 9E9, 9E9, 9E9, 9E9, 9E9]];
	VAR jointtarget CDP_4247 := [[-11.86, 35.68, 6.07, 0, 48.25, -123.66], [9E9, 9E9, 9E9, 9E9, 9E9, 9E9]];
	VAR jointtarget CDP_4248 := [[-11.85, 35.67, 6.08, 0, 48.25, -123.65], [9E9, 9E9, 9E9, 9E9, 9E9, 9E9]];
	VAR jointtarget CDP_4249 := [[-11.84, 35.66, 6.09, 0, 48.24, -123.64], [9E9, 9E9, 9E9, 9E9, 9E9, 9E9]];
	VAR jointtarget CDP_4250 := [[-11.83, 35.65, 6.11, 0, 48.24, -123.63], [9E9, 9E9, 9E9, 9E9, 9E9, 9E9]];
	VAR jointtarget CDP_4251 := [[-11.82, 35.65, 6.12, 0, 48.24, -123.62], [9E9, 9E9, 9E9, 9E9, 9E9, 9E9]];
	VAR jointtarget CDP_4252 := [[-11.81, 35.64, 6.13, 0, 48.23, -123.61], [9E9, 9E9, 9E9, 9E9, 9E9, 9E9]];
	VAR jointtarget CDP_4253 := [[-11.8, 35.63, 6.14, 0, 48.23, -123.6], [9E9, 9E9, 9E9, 9E9, 9E9, 9E9]];
	VAR jointtarget CDP_4254 := [[-11.79, 35.62, 6.16, 0, 48.22, -123.59], [9E9, 9E9, 9E9, 9E9, 9E9, 9E9]];
	VAR jointtarget CDP_4255 := [[-11.78, 35.61, 6.17, 0, 48.22, -123.58], [9E9, 9E9, 9E9, 9E9, 9E9, 9E9]];
	VAR jointtarget CDP_4256 := [[-11.77, 35.61, 6.18, 0, 48.21, -123.57], [9E9, 9E9, 9E9, 9E9, 9E9, 9E9]];
	VAR jointtarget CDP_4257 := [[-11.76, 35.6, 6.19, 0, 48.21, -123.56], [9E9, 9E9, 9E9, 9E9, 9E9, 9E9]];
	VAR jointtarget CDP_4258 := [[-11.75, 35.59, 6.21, 0, 48.2, -123.55], [9E9, 9E9, 9E9, 9E9, 9E9, 9E9]];
	VAR jointtarget CDP_4259 := [[-11.74, 35.58, 6.22, 0, 48.2, -123.54], [9E9, 9E9, 9E9, 9E9, 9E9, 9E9]];
	VAR jointtarget CDP_4260 := [[-10.65, 35.35, 6.62, 0, 48.03, -100.65], [9E9, 9E9, 9E9, 9E9, 9E9, 9E9]];
	VAR jointtarget CDP_4261 := [[-9.55, 35.14, 6.97, 0, 47.88, -99.55], [9E9, 9E9, 9E9, 9E9, 9E9, 9E9]];
	VAR jointtarget CDP_4262 := [[-8.44, 34.95, 7.29, 0, 47.75, -98.44], [9E9, 9E9, 9E9, 9E9, 9E9, 9E9]];
	VAR jointtarget CDP_4263 := [[-7.33, 34.79, 7.57, 0, 47.64, -97.33], [9E9, 9E9, 9E9, 9E9, 9E9, 9E9]];
	VAR jointtarget CDP_4264 := [[-6.21, 34.65, 7.81, 0, 47.54, -96.21], [9E9, 9E9, 9E9, 9E9, 9E9, 9E9]];
	VAR jointtarget CDP_4265 := [[-5.09, 34.53, 8.01, 0, 47.46, -95.09], [9E9, 9E9, 9E9, 9E9, 9E9, 9E9]];
	VAR jointtarget CDP_4266 := [[-3.96, 34.44, 8.17, 0, 47.39, -93.96], [9E9, 9E9, 9E9, 9E9, 9E9, 9E9]];
	VAR jointtarget CDP_4267 := [[-2.83, 34.37, 8.29, 0, 47.34, -92.83], [9E9, 9E9, 9E9, 9E9, 9E9, 9E9]];
	VAR jointtarget CDP_4268 := [[-1.7, 34.32, 8.37, 0, 47.31, -91.7], [9E9, 9E9, 9E9, 9E9, 9E9, 9E9]];
	VAR jointtarget CDP_4269 := [[-0.56, 34.3, 8.41, 0, 47.3, -90.56], [9E9, 9E9, 9E9, 9E9, 9E9, 9E9]];
	VAR jointtarget CDP_4270 := [[0.57, 34.3, 8.41, 0, 47.3, -89.43], [9E9, 9E9, 9E9, 9E9, 9E9, 9E9]];
	VAR jointtarget CDP_4271 := [[1.7, 34.32, 8.37, 0, 47.31, -88.3], [9E9, 9E9, 9E9, 9E9, 9E9, 9E9]];
	VAR jointtarget CDP_4272 := [[2.84, 34.37, 8.29, 0, 47.35, -87.16], [9E9, 9E9, 9E9, 9E9, 9E9, 9E9]];
	VAR jointtarget CDP_4273 := [[3.97, 34.44, 8.17, 0, 47.39, -86.03], [9E9, 9E9, 9E9, 9E9, 9E9, 9E9]];
	VAR jointtarget CDP_4274 := [[5.09, 34.53, 8.01, 0, 47.46, -84.91], [9E9, 9E9, 9E9, 9E9, 9E9, 9E9]];
	VAR jointtarget CDP_4275 := [[6.22, 34.65, 7.81, 0, 47.54, -83.78], [9E9, 9E9, 9E9, 9E9, 9E9, 9E9]];
	VAR jointtarget CDP_4276 := [[7.34, 34.79, 7.57, 0, 47.64, -82.66], [9E9, 9E9, 9E9, 9E9, 9E9, 9E9]];
	VAR jointtarget CDP_4277 := [[8.45, 34.95, 7.29, 0, 47.75, -81.55], [9E9, 9E9, 9E9, 9E9, 9E9, 9E9]];
	VAR jointtarget CDP_4278 := [[9.56, 35.14, 6.97, 0, 47.89, -80.44], [9E9, 9E9, 9E9, 9E9, 9E9, 9E9]];
	VAR jointtarget CDP_4279 := [[10.65, 35.35, 6.61, 0, 48.03, -79.35], [9E9, 9E9, 9E9, 9E9, 9E9, 9E9]];
	VAR jointtarget CDP_4280 := [[10.71, 35.36, 6.59, 0, 48.04, -78.19], [9E9, 9E9, 9E9, 9E9, 9E9, 9E9]];
	VAR jointtarget CDP_4281 := [[10.76, 35.38, 6.57, 0, 48.05, -75.95], [9E9, 9E9, 9E9, 9E9, 9E9, 9E9]];
	VAR jointtarget CDP_4282 := [[10.82, 35.4, 6.54, 0, 48.06, -73.7], [9E9, 9E9, 9E9, 9E9, 9E9, 9E9]];
	VAR jointtarget CDP_4283 := [[10.87, 35.41, 6.51, 0, 48.08, -71.45], [9E9, 9E9, 9E9, 9E9, 9E9, 9E9]];
	VAR jointtarget CDP_4284 := [[10.92, 35.44, 6.47, 0, 48.09, -69.2], [9E9, 9E9, 9E9, 9E9, 9E9, 9E9]];
	VAR jointtarget CDP_4285 := [[10.97, 35.46, 6.43, 0, 48.11, -66.96], [9E9, 9E9, 9E9, 9E9, 9E9, 9E9]];
	VAR jointtarget CDP_4286 := [[11.03, 35.49, 6.39, 0, 48.13, -64.72], [9E9, 9E9, 9E9, 9E9, 9E9, 9E9]];
	VAR jointtarget CDP_4287 := [[11.07, 35.51, 6.34, 0, 48.15, -62.47], [9E9, 9E9, 9E9, 9E9, 9E9, 9E9]];
	VAR jointtarget CDP_4288 := [[11.12, 35.54, 6.29, 0, 48.17, -60.23], [9E9, 9E9, 9E9, 9E9, 9E9, 9E9]];
	VAR jointtarget CDP_4289 := [[11.17, 35.57, 6.23, 0, 48.19, -57.99], [9E9, 9E9, 9E9, 9E9, 9E9, 9E9]];
	VAR jointtarget CDP_4290 := [[11.22, 35.61, 6.18, 0, 48.22, -55.75], [9E9, 9E9, 9E9, 9E9, 9E9, 9E9]];
	VAR jointtarget CDP_4291 := [[11.26, 35.64, 6.11, 0, 48.24, -53.51], [9E9, 9E9, 9E9, 9E9, 9E9, 9E9]];
	VAR jointtarget CDP_4292 := [[11.3, 35.68, 6.05, 0, 48.27, -51.27], [9E9, 9E9, 9E9, 9E9, 9E9, 9E9]];
	VAR jointtarget CDP_4293 := [[11.35, 35.72, 5.98, 0, 48.3, -49.04], [9E9, 9E9, 9E9, 9E9, 9E9, 9E9]];
	VAR jointtarget CDP_4294 := [[11.39, 35.76, 5.91, 0, 48.32, -46.8], [9E9, 9E9, 9E9, 9E9, 9E9, 9E9]];
	VAR jointtarget CDP_4295 := [[11.43, 35.81, 5.84, 0, 48.36, -44.57], [9E9, 9E9, 9E9, 9E9, 9E9, 9E9]];
	VAR jointtarget CDP_4296 := [[11.46, 35.85, 5.76, 0, 48.39, -42.34], [9E9, 9E9, 9E9, 9E9, 9E9, 9E9]];
	VAR jointtarget CDP_4297 := [[11.5, 35.9, 5.68, 0, 48.42, -40.11], [9E9, 9E9, 9E9, 9E9, 9E9, 9E9]];
	VAR jointtarget CDP_4298 := [[11.53, 35.94, 5.6, 0, 48.45, -37.88], [9E9, 9E9, 9E9, 9E9, 9E9, 9E9]];
	VAR jointtarget CDP_4299 := [[11.57, 35.99, 5.52, 0, 48.49, -35.65], [9E9, 9E9, 9E9, 9E9, 9E9, 9E9]];
	VAR jointtarget CDP_4300 := [[11.59, 36.02, 5.47, 0, 48.51, -34.54], [9E9, 9E9, 9E9, 9E9, 9E9, 9E9]];
	VAR jointtarget CDP_4301 := [[11.6, 36.05, 5.41, 0, 48.53, -34.52], [9E9, 9E9, 9E9, 9E9, 9E9, 9E9]];
	VAR jointtarget CDP_4302 := [[11.62, 36.08, 5.36, 0, 48.55, -34.5], [9E9, 9E9, 9E9, 9E9, 9E9, 9E9]];
	VAR jointtarget CDP_4303 := [[11.64, 36.11, 5.31, 0, 48.57, -34.48], [9E9, 9E9, 9E9, 9E9, 9E9, 9E9]];
	VAR jointtarget CDP_4304 := [[11.66, 36.14, 5.26, 0, 48.6, -34.46], [9E9, 9E9, 9E9, 9E9, 9E9, 9E9]];
	VAR jointtarget CDP_4305 := [[11.68, 36.17, 5.21, 0, 48.62, -34.44], [9E9, 9E9, 9E9, 9E9, 9E9, 9E9]];
	VAR jointtarget CDP_4306 := [[11.7, 36.2, 5.16, 0, 48.64, -34.42], [9E9, 9E9, 9E9, 9E9, 9E9, 9E9]];
	VAR jointtarget CDP_4307 := [[11.72, 36.24, 5.1, 0, 48.66, -34.41], [9E9, 9E9, 9E9, 9E9, 9E9, 9E9]];
	VAR jointtarget CDP_4308 := [[11.74, 36.27, 5.05, 0, 48.68, -34.39], [9E9, 9E9, 9E9, 9E9, 9E9, 9E9]];
	VAR jointtarget CDP_4309 := [[11.76, 36.3, 5, 0, 48.7, -34.37], [9E9, 9E9, 9E9, 9E9, 9E9, 9E9]];
	VAR jointtarget CDP_4310 := [[11.77, 36.33, 4.95, 0, 48.73, -34.35], [9E9, 9E9, 9E9, 9E9, 9E9, 9E9]];
	VAR jointtarget CDP_4311 := [[11.79, 36.36, 4.9, 0, 48.75, -34.33], [9E9, 9E9, 9E9, 9E9, 9E9, 9E9]];
	VAR jointtarget CDP_4312 := [[11.81, 36.39, 4.84, 0, 48.77, -34.31], [9E9, 9E9, 9E9, 9E9, 9E9, 9E9]];
	VAR jointtarget CDP_4313 := [[11.83, 36.42, 4.79, 0, 48.79, -34.29], [9E9, 9E9, 9E9, 9E9, 9E9, 9E9]];
	VAR jointtarget CDP_4314 := [[11.85, 36.45, 4.74, 0, 48.81, -34.27], [9E9, 9E9, 9E9, 9E9, 9E9, 9E9]];
	VAR jointtarget CDP_4315 := [[11.87, 36.48, 4.69, 0, 48.83, -34.26], [9E9, 9E9, 9E9, 9E9, 9E9, 9E9]];
	VAR jointtarget CDP_4316 := [[11.89, 36.51, 4.64, 0, 48.86, -34.24], [9E9, 9E9, 9E9, 9E9, 9E9, 9E9]];
	VAR jointtarget CDP_4317 := [[11.91, 36.54, 4.58, 0, 48.88, -34.22], [9E9, 9E9, 9E9, 9E9, 9E9, 9E9]];
	VAR jointtarget CDP_4318 := [[11.92, 36.57, 4.53, 0, 48.9, -34.2], [9E9, 9E9, 9E9, 9E9, 9E9, 9E9]];
	VAR jointtarget CDP_4319 := [[11.94, 36.6, 4.48, 0, 48.92, -34.18], [9E9, 9E9, 9E9, 9E9, 9E9, 9E9]];
	VAR jointtarget CDP_4320 := [[12.05, 36.73, 4.25, 0, 49.02, -40.77], [9E9, 9E9, 9E9, 9E9, 9E9, 9E9]];
	VAR jointtarget CDP_4321 := [[12.18, 36.84, 4.06, 0, 49.09, -54.03], [9E9, 9E9, 9E9, 9E9, 9E9, 9E9]];
	VAR jointtarget CDP_4322 := [[12.33, 36.91, 3.95, 0, 49.14, -67.26], [9E9, 9E9, 9E9, 9E9, 9E9, 9E9]];
	VAR jointtarget CDP_4323 := [[12.49, 36.94, 3.89, 0, 49.17, -80.49], [9E9, 9E9, 9E9, 9E9, 9E9, 9E9]];
	VAR jointtarget CDP_4324 := [[12.65, 36.93, 3.92, 0, 49.16, -93.72], [9E9, 9E9, 9E9, 9E9, 9E9, 9E9]];
	VAR jointtarget CDP_4325 := [[12.8, 36.87, 4.01, 0, 49.12, -106.95], [9E9, 9E9, 9E9, 9E9, 9E9, 9E9]];
	VAR jointtarget CDP_4326 := [[12.94, 36.78, 4.16, 0, 49.05, -120.2], [9E9, 9E9, 9E9, 9E9, 9E9, 9E9]];
	VAR jointtarget CDP_4327 := [[13.06, 36.66, 4.38, 0, 48.96, -133.47], [9E9, 9E9, 9E9, 9E9, 9E9, 9E9]];
	VAR jointtarget CDP_4328 := [[13.15, 36.51, 4.63, 0, 48.86, -146.77], [9E9, 9E9, 9E9, 9E9, 9E9, 9E9]];
	VAR jointtarget CDP_4329 := [[13.2, 36.34, 4.92, 0, 48.74, -160.1], [9E9, 9E9, 9E9, 9E9, 9E9, 9E9]];
	VAR jointtarget CDP_4330 := [[13.22, 36.16, 5.23, 0, 48.61, -173.47], [9E9, 9E9, 9E9, 9E9, 9E9, 9E9]];
	VAR jointtarget CDP_4331 := [[13.2, 35.99, 5.53, 0, 48.48, -186.88], [9E9, 9E9, 9E9, 9E9, 9E9, 9E9]];
	VAR jointtarget CDP_4332 := [[13.15, 35.82, 5.82, 0, 48.36, -200.32], [9E9, 9E9, 9E9, 9E9, 9E9, 9E9]];
	VAR jointtarget CDP_4333 := [[13.06, 35.67, 6.07, 0, 48.26, -213.8], [9E9, 9E9, 9E9, 9E9, 9E9, 9E9]];
	VAR jointtarget CDP_4334 := [[12.93, 35.55, 6.28, 0, 48.17, -227.31], [9E9, 9E9, 9E9, 9E9, 9E9, 9E9]];
	VAR jointtarget CDP_4335 := [[12.79, 35.46, 6.43, 0, 48.11, -240.84], [9E9, 9E9, 9E9, 9E9, 9E9, 9E9]];
	VAR jointtarget CDP_4336 := [[12.63, 35.41, 6.51, 0, 48.08, -254.39], [9E9, 9E9, 9E9, 9E9, 9E9, 9E9]];
	VAR jointtarget CDP_4337 := [[12.47, 35.41, 6.52, 0, 48.07, -267.94], [9E9, 9E9, 9E9, 9E9, 9E9, 9E9]];
	VAR jointtarget CDP_4338 := [[12.3, 35.44, 6.46, 0, 48.1, -281.49], [9E9, 9E9, 9E9, 9E9, 9E9, 9E9]];
	VAR jointtarget CDP_4339 := [[12.15, 35.52, 6.33, 0, 48.15, -295.03], [9E9, 9E9, 9E9, 9E9, 9E9, 9E9]];
	VAR jointtarget CDP_4340 := [[12.13, 35.54, 6.3, 0, 48.16, -301.75], [9E9, 9E9, 9E9, 9E9, 9E9, 9E9]];
	VAR jointtarget CDP_4341 := [[12.1, 35.56, 6.27, 0, 48.18, -301.78], [9E9, 9E9, 9E9, 9E9, 9E9, 9E9]];
	VAR jointtarget CDP_4342 := [[12.07, 35.57, 6.23, 0, 48.19, -301.81], [9E9, 9E9, 9E9, 9E9, 9E9, 9E9]];
	VAR jointtarget CDP_4343 := [[12.04, 35.59, 6.2, 0, 48.2, -301.84], [9E9, 9E9, 9E9, 9E9, 9E9, 9E9]];
	VAR jointtarget CDP_4344 := [[12.01, 35.61, 6.17, 0, 48.22, -301.87], [9E9, 9E9, 9E9, 9E9, 9E9, 9E9]];
	VAR jointtarget CDP_4345 := [[11.98, 35.63, 6.14, 0, 48.23, -301.89], [9E9, 9E9, 9E9, 9E9, 9E9, 9E9]];
	VAR jointtarget CDP_4346 := [[11.95, 35.65, 6.1, 0, 48.25, -301.92], [9E9, 9E9, 9E9, 9E9, 9E9, 9E9]];
	VAR jointtarget CDP_4347 := [[11.92, 35.67, 6.07, 0, 48.26, -301.95], [9E9, 9E9, 9E9, 9E9, 9E9, 9E9]];
	VAR jointtarget CDP_4348 := [[11.9, 35.69, 6.04, 0, 48.27, -301.98], [9E9, 9E9, 9E9, 9E9, 9E9, 9E9]];
	VAR jointtarget CDP_4349 := [[11.87, 35.71, 6, 0, 48.29, -302.01], [9E9, 9E9, 9E9, 9E9, 9E9, 9E9]];
	VAR jointtarget CDP_4350 := [[11.84, 35.73, 5.97, 0, 48.3, -302.04], [9E9, 9E9, 9E9, 9E9, 9E9, 9E9]];
	VAR jointtarget CDP_4351 := [[11.81, 35.75, 5.94, 0, 48.31, -302.07], [9E9, 9E9, 9E9, 9E9, 9E9, 9E9]];
	VAR jointtarget CDP_4352 := [[11.78, 35.77, 5.91, 0, 48.33, -302.09], [9E9, 9E9, 9E9, 9E9, 9E9, 9E9]];
	VAR jointtarget CDP_4353 := [[11.75, 35.79, 5.87, 0, 48.34, -302.12], [9E9, 9E9, 9E9, 9E9, 9E9, 9E9]];
	VAR jointtarget CDP_4354 := [[11.73, 35.81, 5.84, 0, 48.36, -302.15], [9E9, 9E9, 9E9, 9E9, 9E9, 9E9]];
	VAR jointtarget CDP_4355 := [[11.7, 35.83, 5.81, 0, 48.37, -302.18], [9E9, 9E9, 9E9, 9E9, 9E9, 9E9]];
	VAR jointtarget CDP_4356 := [[11.67, 35.84, 5.77, 0, 48.38, -302.21], [9E9, 9E9, 9E9, 9E9, 9E9, 9E9]];
	VAR jointtarget CDP_4357 := [[11.64, 35.86, 5.74, 0, 48.4, -302.24], [9E9, 9E9, 9E9, 9E9, 9E9, 9E9]];
	VAR jointtarget CDP_4358 := [[11.61, 35.88, 5.71, 0, 48.41, -302.27], [9E9, 9E9, 9E9, 9E9, 9E9, 9E9]];
	VAR jointtarget CDP_4359 := [[11.58, 35.9, 5.67, 0, 48.42, -302.29], [9E9, 9E9, 9E9, 9E9, 9E9, 9E9]];
	VAR jointtarget CDP_4360 := [[11.54, 35.93, 5.62, 0, 48.45, -301.24], [9E9, 9E9, 9E9, 9E9, 9E9, 9E9]];
	VAR jointtarget CDP_4361 := [[11.49, 35.96, 5.57, 0, 48.47, -299.1], [9E9, 9E9, 9E9, 9E9, 9E9, 9E9]];
	VAR jointtarget CDP_4362 := [[11.44, 35.99, 5.52, 0, 48.49, -296.95], [9E9, 9E9, 9E9, 9E9, 9E9, 9E9]];
	VAR jointtarget CDP_4363 := [[11.39, 36.02, 5.48, 0, 48.51, -294.81], [9E9, 9E9, 9E9, 9E9, 9E9, 9E9]];
	VAR jointtarget CDP_4364 := [[11.34, 36.04, 5.44, 0, 48.52, -292.67], [9E9, 9E9, 9E9, 9E9, 9E9, 9E9]];
	VAR jointtarget CDP_4365 := [[11.28, 36.06, 5.4, 0, 48.54, -290.53], [9E9, 9E9, 9E9, 9E9, 9E9, 9E9]];
	VAR jointtarget CDP_4366 := [[11.23, 36.08, 5.37, 0, 48.55, -288.38], [9E9, 9E9, 9E9, 9E9, 9E9, 9E9]];
	VAR jointtarget CDP_4367 := [[11.18, 36.1, 5.34, 0, 48.56, -286.24], [9E9, 9E9, 9E9, 9E9, 9E9, 9E9]];
	VAR jointtarget CDP_4368 := [[11.13, 36.11, 5.32, 0, 48.57, -284.1], [9E9, 9E9, 9E9, 9E9, 9E9, 9E9]];
	VAR jointtarget CDP_4369 := [[11.07, 36.12, 5.29, 0, 48.58, -281.96], [9E9, 9E9, 9E9, 9E9, 9E9, 9E9]];
	VAR jointtarget CDP_4370 := [[11.02, 36.13, 5.28, 0, 48.59, -279.82], [9E9, 9E9, 9E9, 9E9, 9E9, 9E9]];
	VAR jointtarget CDP_4371 := [[10.96, 36.14, 5.26, 0, 48.59, -277.69], [9E9, 9E9, 9E9, 9E9, 9E9, 9E9]];
	VAR jointtarget CDP_4372 := [[10.91, 36.15, 5.25, 0, 48.6, -275.55], [9E9, 9E9, 9E9, 9E9, 9E9, 9E9]];
	VAR jointtarget CDP_4373 := [[10.85, 36.15, 5.25, 0, 48.6, -273.41], [9E9, 9E9, 9E9, 9E9, 9E9, 9E9]];
	VAR jointtarget CDP_4374 := [[10.8, 36.15, 5.24, 0, 48.6, -271.27], [9E9, 9E9, 9E9, 9E9, 9E9, 9E9]];
	VAR jointtarget CDP_4375 := [[10.74, 36.15, 5.25, 0, 48.6, -269.13], [9E9, 9E9, 9E9, 9E9, 9E9, 9E9]];
	VAR jointtarget CDP_4376 := [[10.69, 36.15, 5.25, 0, 48.6, -266.99], [9E9, 9E9, 9E9, 9E9, 9E9, 9E9]];
	VAR jointtarget CDP_4377 := [[10.63, 36.14, 5.26, 0, 48.6, -264.85], [9E9, 9E9, 9E9, 9E9, 9E9, 9E9]];
	VAR jointtarget CDP_4378 := [[10.58, 36.14, 5.27, 0, 48.59, -262.71], [9E9, 9E9, 9E9, 9E9, 9E9, 9E9]];
	VAR jointtarget CDP_4379 := [[10.52, 36.13, 5.29, 0, 48.58, -260.58], [9E9, 9E9, 9E9, 9E9, 9E9, 9E9]];
	VAR jointtarget CDP_4380 := [[9.44, 35.92, 5.65, 0, 48.44, -260.56], [9E9, 9E9, 9E9, 9E9, 9E9, 9E9]];
	VAR jointtarget CDP_4381 := [[8.36, 35.73, 5.96, 0, 48.3, -261.64], [9E9, 9E9, 9E9, 9E9, 9E9, 9E9]];
	VAR jointtarget CDP_4382 := [[7.27, 35.57, 6.24, 0, 48.19, -262.73], [9E9, 9E9, 9E9, 9E9, 9E9, 9E9]];
	VAR jointtarget CDP_4383 := [[6.17, 35.43, 6.48, 0, 48.09, -263.83], [9E9, 9E9, 9E9, 9E9, 9E9, 9E9]];
	VAR jointtarget CDP_4384 := [[5.07, 35.32, 6.67, 0, 48.01, -264.93], [9E9, 9E9, 9E9, 9E9, 9E9, 9E9]];
	VAR jointtarget CDP_4385 := [[3.97, 35.22, 6.83, 0, 47.94, -266.03], [9E9, 9E9, 9E9, 9E9, 9E9, 9E9]];
	VAR jointtarget CDP_4386 := [[2.86, 35.15, 6.95, 0, 47.89, -267.14], [9E9, 9E9, 9E9, 9E9, 9E9, 9E9]];
	VAR jointtarget CDP_4387 := [[1.75, 35.1, 7.04, 0, 47.86, -268.25], [9E9, 9E9, 9E9, 9E9, 9E9, 9E9]];
	VAR jointtarget CDP_4388 := [[0.64, 35.08, 7.08, 0, 47.84, -269.36], [9E9, 9E9, 9E9, 9E9, 9E9, 9E9]];
	VAR jointtarget CDP_4389 := [[-0.47, 35.08, 7.08, 0, 47.84, -270.47], [9E9, 9E9, 9E9, 9E9, 9E9, 9E9]];
	VAR jointtarget CDP_4390 := [[-1.58, 35.1, 7.04, 0, 47.86, -271.58], [9E9, 9E9, 9E9, 9E9, 9E9, 9E9]];
	VAR jointtarget CDP_4391 := [[-2.69, 35.14, 6.97, 0, 47.89, -272.69], [9E9, 9E9, 9E9, 9E9, 9E9, 9E9]];
	VAR jointtarget CDP_4392 := [[-3.8, 35.21, 6.85, 0, 47.93, -273.8], [9E9, 9E9, 9E9, 9E9, 9E9, 9E9]];
	VAR jointtarget CDP_4393 := [[-4.9, 35.3, 6.7, 0, 48, -274.9], [9E9, 9E9, 9E9, 9E9, 9E9, 9E9]];
	VAR jointtarget CDP_4394 := [[-6, 35.41, 6.51, 0, 48.08, -276], [9E9, 9E9, 9E9, 9E9, 9E9, 9E9]];
	VAR jointtarget CDP_4395 := [[-7.1, 35.55, 6.28, 0, 48.17, -277.1], [9E9, 9E9, 9E9, 9E9, 9E9, 9E9]];
	VAR jointtarget CDP_4396 := [[-8.19, 35.71, 6.01, 0, 48.29, -278.19], [9E9, 9E9, 9E9, 9E9, 9E9, 9E9]];
	VAR jointtarget CDP_4397 := [[-9.28, 35.89, 5.7, 0, 48.41, -279.28], [9E9, 9E9, 9E9, 9E9, 9E9, 9E9]];
	VAR jointtarget CDP_4398 := [[-10.36, 36.09, 5.35, 0, 48.56, -280.36], [9E9, 9E9, 9E9, 9E9, 9E9, 9E9]];
	VAR jointtarget CDP_4399 := [[-11.43, 36.32, 4.96, 0, 48.72, -281.43], [9E9, 9E9, 9E9, 9E9, 9E9, 9E9]];
	VAR jointtarget CDP_4400 := [[-11.44, 36.32, 4.95, 0, 48.72, -281.78], [9E9, 9E9, 9E9, 9E9, 9E9, 9E9]];
	VAR jointtarget CDP_4401 := [[-11.46, 36.33, 4.95, 0, 48.73, -282.45], [9E9, 9E9, 9E9, 9E9, 9E9, 9E9]];
	VAR jointtarget CDP_4402 := [[-11.48, 36.33, 4.94, 0, 48.73, -283.13], [9E9, 9E9, 9E9, 9E9, 9E9, 9E9]];
	VAR jointtarget CDP_4403 := [[-11.49, 36.34, 4.93, 0, 48.73, -283.81], [9E9, 9E9, 9E9, 9E9, 9E9, 9E9]];
	VAR jointtarget CDP_4404 := [[-11.51, 36.34, 4.92, 0, 48.74, -284.49], [9E9, 9E9, 9E9, 9E9, 9E9, 9E9]];
	VAR jointtarget CDP_4405 := [[-11.53, 36.35, 4.92, 0, 48.74, -285.17], [9E9, 9E9, 9E9, 9E9, 9E9, 9E9]];
	VAR jointtarget CDP_4406 := [[-11.54, 36.35, 4.91, 0, 48.74, -285.84], [9E9, 9E9, 9E9, 9E9, 9E9, 9E9]];
	VAR jointtarget CDP_4407 := [[-11.56, 36.36, 4.9, 0, 48.75, -286.52], [9E9, 9E9, 9E9, 9E9, 9E9, 9E9]];
	VAR jointtarget CDP_4408 := [[-11.57, 36.36, 4.89, 0, 48.75, -287.2], [9E9, 9E9, 9E9, 9E9, 9E9, 9E9]];
	VAR jointtarget CDP_4409 := [[-11.59, 36.37, 4.88, 0, 48.75, -287.88], [9E9, 9E9, 9E9, 9E9, 9E9, 9E9]];
	VAR jointtarget CDP_4410 := [[-11.6, 36.37, 4.87, 0, 48.76, -288.56], [9E9, 9E9, 9E9, 9E9, 9E9, 9E9]];
	VAR jointtarget CDP_4411 := [[-11.62, 36.38, 4.86, 0, 48.76, -289.23], [9E9, 9E9, 9E9, 9E9, 9E9, 9E9]];
	VAR jointtarget CDP_4412 := [[-11.64, 36.38, 4.85, 0, 48.77, -289.91], [9E9, 9E9, 9E9, 9E9, 9E9, 9E9]];
	VAR jointtarget CDP_4413 := [[-11.65, 36.39, 4.84, 0, 48.77, -290.59], [9E9, 9E9, 9E9, 9E9, 9E9, 9E9]];
	VAR jointtarget CDP_4414 := [[-11.67, 36.4, 4.83, 0, 48.78, -291.27], [9E9, 9E9, 9E9, 9E9, 9E9, 9E9]];
	VAR jointtarget CDP_4415 := [[-11.68, 36.4, 4.81, 0, 48.78, -291.94], [9E9, 9E9, 9E9, 9E9, 9E9, 9E9]];
	VAR jointtarget CDP_4416 := [[-11.7, 36.41, 4.8, 0, 48.79, -292.62], [9E9, 9E9, 9E9, 9E9, 9E9, 9E9]];
	VAR jointtarget CDP_4417 := [[-11.71, 36.42, 4.79, 0, 48.79, -293.3], [9E9, 9E9, 9E9, 9E9, 9E9, 9E9]];
	VAR jointtarget CDP_4418 := [[-11.73, 36.43, 4.78, 0, 48.8, -293.98], [9E9, 9E9, 9E9, 9E9, 9E9, 9E9]];
	VAR jointtarget CDP_4419 := [[-11.74, 36.43, 4.76, 0, 48.8, -294.65], [9E9, 9E9, 9E9, 9E9, 9E9, 9E9]];
	VAR jointtarget CDP_4420 := [[-11.8, 36.46, 4.71, 0, 48.82, -295.04], [9E9, 9E9, 9E9, 9E9, 9E9, 9E9]];
	VAR jointtarget CDP_4421 := [[-11.86, 36.5, 4.66, 0, 48.85, -295.11], [9E9, 9E9, 9E9, 9E9, 9E9, 9E9]];
	VAR jointtarget CDP_4422 := [[-11.93, 36.53, 4.6, 0, 48.87, -295.17], [9E9, 9E9, 9E9, 9E9, 9E9, 9E9]];
	VAR jointtarget CDP_4423 := [[-11.99, 36.56, 4.55, 0, 48.89, -295.23], [9E9, 9E9, 9E9, 9E9, 9E9, 9E9]];
	VAR jointtarget CDP_4424 := [[-12.05, 36.59, 4.49, 0, 48.92, -295.29], [9E9, 9E9, 9E9, 9E9, 9E9, 9E9]];
	VAR jointtarget CDP_4425 := [[-12.11, 36.62, 4.44, 0, 48.94, -295.35], [9E9, 9E9, 9E9, 9E9, 9E9, 9E9]];
	VAR jointtarget CDP_4426 := [[-12.17, 36.65, 4.39, 0, 48.96, -295.41], [9E9, 9E9, 9E9, 9E9, 9E9, 9E9]];
	VAR jointtarget CDP_4427 := [[-12.23, 36.69, 4.33, 0, 48.98, -295.47], [9E9, 9E9, 9E9, 9E9, 9E9, 9E9]];
	VAR jointtarget CDP_4428 := [[-12.29, 36.72, 4.28, 0, 49.01, -295.53], [9E9, 9E9, 9E9, 9E9, 9E9, 9E9]];
	VAR jointtarget CDP_4429 := [[-12.35, 36.75, 4.22, 0, 49.03, -295.59], [9E9, 9E9, 9E9, 9E9, 9E9, 9E9]];
	VAR jointtarget CDP_4430 := [[-12.41, 36.78, 4.17, 0, 49.05, -295.65], [9E9, 9E9, 9E9, 9E9, 9E9, 9E9]];
	VAR jointtarget CDP_4431 := [[-12.47, 36.81, 4.11, 0, 49.08, -295.71], [9E9, 9E9, 9E9, 9E9, 9E9, 9E9]];
	VAR jointtarget CDP_4432 := [[-12.53, 36.85, 4.06, 0, 49.1, -295.77], [9E9, 9E9, 9E9, 9E9, 9E9, 9E9]];
	VAR jointtarget CDP_4433 := [[-12.59, 36.88, 4, 0, 49.12, -295.83], [9E9, 9E9, 9E9, 9E9, 9E9, 9E9]];
	VAR jointtarget CDP_4434 := [[-12.65, 36.91, 3.94, 0, 49.15, -295.89], [9E9, 9E9, 9E9, 9E9, 9E9, 9E9]];
	VAR jointtarget CDP_4435 := [[-12.71, 36.94, 3.89, 0, 49.17, -295.95], [9E9, 9E9, 9E9, 9E9, 9E9, 9E9]];
	VAR jointtarget CDP_4436 := [[-12.77, 36.98, 3.83, 0, 49.19, -296.01], [9E9, 9E9, 9E9, 9E9, 9E9, 9E9]];
	VAR jointtarget CDP_4437 := [[-12.83, 37.01, 3.78, 0, 49.22, -296.07], [9E9, 9E9, 9E9, 9E9, 9E9, 9E9]];
	VAR jointtarget CDP_4438 := [[-12.89, 37.04, 3.72, 0, 49.24, -296.13], [9E9, 9E9, 9E9, 9E9, 9E9, 9E9]];
	VAR jointtarget CDP_4439 := [[-12.95, 37.07, 3.66, 0, 49.26, -296.19], [9E9, 9E9, 9E9, 9E9, 9E9, 9E9]];
	VAR jointtarget CDP_4440 := [[-13.07, 37.13, 3.57, 0, 49.3, -291.14], [9E9, 9E9, 9E9, 9E9, 9E9, 9E9]];
	VAR jointtarget CDP_4441 := [[-13.19, 37.15, 3.53, 0, 49.32, -280.95], [9E9, 9E9, 9E9, 9E9, 9E9, 9E9]];
	VAR jointtarget CDP_4442 := [[-13.32, 37.15, 3.52, 0, 49.32, -270.75], [9E9, 9E9, 9E9, 9E9, 9E9, 9E9]];
	VAR jointtarget CDP_4443 := [[-13.45, 37.13, 3.57, 0, 49.3, -260.55], [9E9, 9E9, 9E9, 9E9, 9E9, 9E9]];
	VAR jointtarget CDP_4444 := [[-13.57, 37.08, 3.65, 0, 49.27, -250.35], [9E9, 9E9, 9E9, 9E9, 9E9, 9E9]];
	VAR jointtarget CDP_4445 := [[-13.68, 37.01, 3.77, 0, 49.22, -240.14], [9E9, 9E9, 9E9, 9E9, 9E9, 9E9]];
	VAR jointtarget CDP_4446 := [[-13.78, 36.92, 3.93, 0, 49.15, -229.91], [9E9, 9E9, 9E9, 9E9, 9E9, 9E9]];
	VAR jointtarget CDP_4447 := [[-13.86, 36.81, 4.12, 0, 49.07, -219.67], [9E9, 9E9, 9E9, 9E9, 9E9, 9E9]];
	VAR jointtarget CDP_4448 := [[-13.93, 36.68, 4.34, 0, 48.98, -209.41], [9E9, 9E9, 9E9, 9E9, 9E9, 9E9]];
	VAR jointtarget CDP_4449 := [[-13.97, 36.54, 4.57, 0, 48.88, -199.13], [9E9, 9E9, 9E9, 9E9, 9E9, 9E9]];
	VAR jointtarget CDP_4450 := [[-13.99, 36.4, 4.82, 0, 48.78, -188.83], [9E9, 9E9, 9E9, 9E9, 9E9, 9E9]];
	VAR jointtarget CDP_4451 := [[-13.98, 36.26, 5.06, 0, 48.68, -178.5], [9E9, 9E9, 9E9, 9E9, 9E9, 9E9]];
	VAR jointtarget CDP_4452 := [[-13.96, 36.12, 5.3, 0, 48.58, -168.15], [9E9, 9E9, 9E9, 9E9, 9E9, 9E9]];
	VAR jointtarget CDP_4453 := [[-13.91, 35.99, 5.53, 0, 48.48, -157.77], [9E9, 9E9, 9E9, 9E9, 9E9, 9E9]];
	VAR jointtarget CDP_4454 := [[-13.84, 35.87, 5.74, 0, 48.4, -147.38], [9E9, 9E9, 9E9, 9E9, 9E9, 9E9]];
	VAR jointtarget CDP_4455 := [[-13.75, 35.76, 5.92, 0, 48.32, -136.97], [9E9, 9E9, 9E9, 9E9, 9E9, 9E9]];
	VAR jointtarget CDP_4456 := [[-13.64, 35.68, 6.06, 0, 48.26, -126.54], [9E9, 9E9, 9E9, 9E9, 9E9, 9E9]];
	VAR jointtarget CDP_4457 := [[-13.52, 35.61, 6.17, 0, 48.22, -116.09], [9E9, 9E9, 9E9, 9E9, 9E9, 9E9]];
	VAR jointtarget CDP_4458 := [[-13.4, 35.57, 6.23, 0, 48.19, -105.64], [9E9, 9E9, 9E9, 9E9, 9E9, 9E9]];
	VAR jointtarget CDP_4459 := [[-13.27, 35.56, 6.26, 0, 48.18, -95.19], [9E9, 9E9, 9E9, 9E9, 9E9, 9E9]];
	VAR jointtarget CDP_4460 := [[-13.2, 35.56, 6.26, 0, 48.18, -89.96], [9E9, 9E9, 9E9, 9E9, 9E9, 9E9]];
	VAR jointtarget CDP_4461 := [[-13.13, 35.56, 6.26, 0, 48.18, -89.89], [9E9, 9E9, 9E9, 9E9, 9E9, 9E9]];
	VAR jointtarget CDP_4462 := [[-13.06, 35.56, 6.26, 0, 48.18, -89.82], [9E9, 9E9, 9E9, 9E9, 9E9, 9E9]];
	VAR jointtarget CDP_4463 := [[-12.99, 35.56, 6.26, 0, 48.19, -89.75], [9E9, 9E9, 9E9, 9E9, 9E9, 9E9]];
	VAR jointtarget CDP_4464 := [[-12.93, 35.56, 6.25, 0, 48.19, -89.69], [9E9, 9E9, 9E9, 9E9, 9E9, 9E9]];
	VAR jointtarget CDP_4465 := [[-12.86, 35.56, 6.25, 0, 48.19, -89.62], [9E9, 9E9, 9E9, 9E9, 9E9, 9E9]];
	VAR jointtarget CDP_4466 := [[-12.79, 35.56, 6.25, 0, 48.19, -89.55], [9E9, 9E9, 9E9, 9E9, 9E9, 9E9]];
	VAR jointtarget CDP_4467 := [[-12.72, 35.56, 6.25, 0, 48.19, -89.48], [9E9, 9E9, 9E9, 9E9, 9E9, 9E9]];
	VAR jointtarget CDP_4468 := [[-12.65, 35.56, 6.25, 0, 48.19, -89.41], [9E9, 9E9, 9E9, 9E9, 9E9, 9E9]];
	VAR jointtarget CDP_4469 := [[-12.59, 35.56, 6.25, 0, 48.19, -89.35], [9E9, 9E9, 9E9, 9E9, 9E9, 9E9]];
	VAR jointtarget CDP_4470 := [[-12.52, 35.56, 6.25, 0, 48.19, -89.28], [9E9, 9E9, 9E9, 9E9, 9E9, 9E9]];
	VAR jointtarget CDP_4471 := [[-12.45, 35.56, 6.25, 0, 48.19, -89.21], [9E9, 9E9, 9E9, 9E9, 9E9, 9E9]];
	VAR jointtarget CDP_4472 := [[-12.38, 35.56, 6.24, 0, 48.2, -89.14], [9E9, 9E9, 9E9, 9E9, 9E9, 9E9]];
	VAR jointtarget CDP_4473 := [[-12.32, 35.56, 6.24, 0, 48.2, -89.07], [9E9, 9E9, 9E9, 9E9, 9E9, 9E9]];
	VAR jointtarget CDP_4474 := [[-12.25, 35.56, 6.24, 0, 48.2, -89.01], [9E9, 9E9, 9E9, 9E9, 9E9, 9E9]];
	VAR jointtarget CDP_4475 := [[-12.18, 35.56, 6.24, 0, 48.2, -88.94], [9E9, 9E9, 9E9, 9E9, 9E9, 9E9]];
	VAR jointtarget CDP_4476 := [[-12.11, 35.56, 6.23, 0, 48.2, -88.87], [9E9, 9E9, 9E9, 9E9, 9E9, 9E9]];
	VAR jointtarget CDP_4477 := [[-12.04, 35.56, 6.23, 0, 48.2, -88.8], [9E9, 9E9, 9E9, 9E9, 9E9, 9E9]];
	VAR jointtarget CDP_4478 := [[-11.98, 35.57, 6.23, 0, 48.21, -88.74], [9E9, 9E9, 9E9, 9E9, 9E9, 9E9]];
	VAR jointtarget CDP_4479 := [[-11.91, 35.57, 6.23, 0, 48.21, -88.67], [9E9, 9E9, 9E9, 9E9, 9E9, 9E9]];
	VAR jointtarget CDP_4480 := [[-11.89, 35.57, 6.23, 0, 48.21, -88.98], [9E9, 9E9, 9E9, 9E9, 9E9, 9E9]];
	VAR jointtarget CDP_4481 := [[-11.87, 35.57, 6.23, 0, 48.21, -89.63], [9E9, 9E9, 9E9, 9E9, 9E9, 9E9]];
	VAR jointtarget CDP_4482 := [[-11.86, 35.57, 6.23, 0, 48.21, -90.27], [9E9, 9E9, 9E9, 9E9, 9E9, 9E9]];
	VAR jointtarget CDP_4483 := [[-11.84, 35.57, 6.23, 0, 48.21, -90.92], [9E9, 9E9, 9E9, 9E9, 9E9, 9E9]];
	VAR jointtarget CDP_4484 := [[-11.82, 35.57, 6.23, 0, 48.21, -91.56], [9E9, 9E9, 9E9, 9E9, 9E9, 9E9]];
	VAR jointtarget CDP_4485 := [[-11.81, 35.56, 6.23, 0, 48.21, -92.21], [9E9, 9E9, 9E9, 9E9, 9E9, 9E9]];
	VAR jointtarget CDP_4486 := [[-11.79, 35.56, 6.23, 0, 48.21, -92.85], [9E9, 9E9, 9E9, 9E9, 9E9, 9E9]];
	VAR jointtarget CDP_4487 := [[-11.77, 35.56, 6.23, 0, 48.21, -93.5], [9E9, 9E9, 9E9, 9E9, 9E9, 9E9]];
	VAR jointtarget CDP_4488 := [[-11.76, 35.56, 6.23, 0, 48.21, -94.14], [9E9, 9E9, 9E9, 9E9, 9E9, 9E9]];
	VAR jointtarget CDP_4489 := [[-11.74, 35.56, 6.24, 0, 48.2, -94.79], [9E9, 9E9, 9E9, 9E9, 9E9, 9E9]];
	VAR jointtarget CDP_4490 := [[-11.72, 35.56, 6.24, 0, 48.2, -95.43], [9E9, 9E9, 9E9, 9E9, 9E9, 9E9]];
	VAR jointtarget CDP_4491 := [[-11.71, 35.56, 6.24, 0, 48.2, -96.08], [9E9, 9E9, 9E9, 9E9, 9E9, 9E9]];
	VAR jointtarget CDP_4492 := [[-11.69, 35.55, 6.25, 0, 48.2, -96.72], [9E9, 9E9, 9E9, 9E9, 9E9, 9E9]];
	VAR jointtarget CDP_4493 := [[-11.67, 35.55, 6.25, 0, 48.2, -97.37], [9E9, 9E9, 9E9, 9E9, 9E9, 9E9]];
	VAR jointtarget CDP_4494 := [[-11.66, 35.55, 6.25, 0, 48.2, -98.01], [9E9, 9E9, 9E9, 9E9, 9E9, 9E9]];
	VAR jointtarget CDP_4495 := [[-11.64, 35.55, 6.26, 0, 48.2, -98.66], [9E9, 9E9, 9E9, 9E9, 9E9, 9E9]];
	VAR jointtarget CDP_4496 := [[-11.62, 35.54, 6.26, 0, 48.19, -99.31], [9E9, 9E9, 9E9, 9E9, 9E9, 9E9]];
	VAR jointtarget CDP_4497 := [[-11.61, 35.54, 6.27, 0, 48.19, -99.95], [9E9, 9E9, 9E9, 9E9, 9E9, 9E9]];
	VAR jointtarget CDP_4498 := [[-11.59, 35.54, 6.27, 0, 48.19, -100.6], [9E9, 9E9, 9E9, 9E9, 9E9, 9E9]];
	VAR jointtarget CDP_4499 := [[-11.57, 35.53, 6.28, 0, 48.19, -101.24], [9E9, 9E9, 9E9, 9E9, 9E9, 9E9]];
	VAR jointtarget CDP_4500 := [[-10.48, 35.3, 6.67, 0, 48.02, -100.48], [9E9, 9E9, 9E9, 9E9, 9E9, 9E9]];
	VAR jointtarget CDP_4501 := [[-9.38, 35.1, 7.02, 0, 47.88, -99.38], [9E9, 9E9, 9E9, 9E9, 9E9, 9E9]];
	VAR jointtarget CDP_4502 := [[-8.27, 34.91, 7.34, 0, 47.75, -98.27], [9E9, 9E9, 9E9, 9E9, 9E9, 9E9]];
	VAR jointtarget CDP_4503 := [[-7.15, 34.75, 7.61, 0, 47.64, -97.15], [9E9, 9E9, 9E9, 9E9, 9E9, 9E9]];
	VAR jointtarget CDP_4504 := [[-6.03, 34.62, 7.84, 0, 47.54, -96.03], [9E9, 9E9, 9E9, 9E9, 9E9, 9E9]];
	VAR jointtarget CDP_4505 := [[-4.9, 34.5, 8.03, 0, 47.46, -94.9], [9E9, 9E9, 9E9, 9E9, 9E9, 9E9]];
	VAR jointtarget CDP_4506 := [[-3.77, 34.41, 8.19, 0, 47.4, -93.77], [9E9, 9E9, 9E9, 9E9, 9E9, 9E9]];
	VAR jointtarget CDP_4507 := [[-2.64, 34.34, 8.3, 0, 47.35, -92.64], [9E9, 9E9, 9E9, 9E9, 9E9, 9E9]];
	VAR jointtarget CDP_4508 := [[-1.51, 34.3, 8.37, 0, 47.32, -91.51], [9E9, 9E9, 9E9, 9E9, 9E9, 9E9]];
	VAR jointtarget CDP_4509 := [[-0.37, 34.28, 8.41, 0, 47.31, -90.37], [9E9, 9E9, 9E9, 9E9, 9E9, 9E9]];
	VAR jointtarget CDP_4510 := [[0.76, 34.29, 8.4, 0, 47.31, -89.24], [9E9, 9E9, 9E9, 9E9, 9E9, 9E9]];
	VAR jointtarget CDP_4511 := [[1.9, 34.31, 8.35, 0, 47.33, -88.1], [9E9, 9E9, 9E9, 9E9, 9E9, 9E9]];
	VAR jointtarget CDP_4512 := [[3.03, 34.37, 8.27, 0, 47.37, -86.97], [9E9, 9E9, 9E9, 9E9, 9E9, 9E9]];
	VAR jointtarget CDP_4513 := [[4.16, 34.44, 8.14, 0, 47.42, -85.84], [9E9, 9E9, 9E9, 9E9, 9E9, 9E9]];
	VAR jointtarget CDP_4514 := [[5.29, 34.54, 7.97, 0, 47.49, -84.71], [9E9, 9E9, 9E9, 9E9, 9E9, 9E9]];
	VAR jointtarget CDP_4515 := [[6.42, 34.66, 7.77, 0, 47.57, -83.58], [9E9, 9E9, 9E9, 9E9, 9E9, 9E9]];
	VAR jointtarget CDP_4516 := [[7.54, 34.81, 7.52, 0, 47.67, -82.46], [9E9, 9E9, 9E9, 9E9, 9E9, 9E9]];
	VAR jointtarget CDP_4517 := [[8.65, 34.97, 7.23, 0, 47.79, -81.35], [9E9, 9E9, 9E9, 9E9, 9E9, 9E9]];
	VAR jointtarget CDP_4518 := [[9.76, 35.17, 6.91, 0, 47.93, -80.24], [9E9, 9E9, 9E9, 9E9, 9E9, 9E9]];
	VAR jointtarget CDP_4519 := [[10.86, 35.38, 6.54, 0, 48.08, -79.14], [9E9, 9E9, 9E9, 9E9, 9E9, 9E9]];
	VAR jointtarget CDP_4520 := [[10.87, 35.38, 6.54, 0, 48.08, -79.46], [9E9, 9E9, 9E9, 9E9, 9E9, 9E9]];
	VAR jointtarget CDP_4521 := [[10.89, 35.39, 6.53, 0, 48.08, -80.1], [9E9, 9E9, 9E9, 9E9, 9E9, 9E9]];
	VAR jointtarget CDP_4522 := [[10.91, 35.39, 6.53, 0, 48.09, -80.75], [9E9, 9E9, 9E9, 9E9, 9E9, 9E9]];
	VAR jointtarget CDP_4523 := [[10.92, 35.39, 6.52, 0, 48.09, -81.39], [9E9, 9E9, 9E9, 9E9, 9E9, 9E9]];
	VAR jointtarget CDP_4524 := [[10.94, 35.39, 6.52, 0, 48.09, -82.04], [9E9, 9E9, 9E9, 9E9, 9E9, 9E9]];
	VAR jointtarget CDP_4525 := [[10.96, 35.4, 6.51, 0, 48.09, -82.68], [9E9, 9E9, 9E9, 9E9, 9E9, 9E9]];
	VAR jointtarget CDP_4526 := [[10.97, 35.4, 6.51, 0, 48.09, -83.33], [9E9, 9E9, 9E9, 9E9, 9E9, 9E9]];
	VAR jointtarget CDP_4527 := [[10.99, 35.4, 6.51, 0, 48.09, -83.97], [9E9, 9E9, 9E9, 9E9, 9E9, 9E9]];
	VAR jointtarget CDP_4528 := [[11.01, 35.4, 6.5, 0, 48.09, -84.62], [9E9, 9E9, 9E9, 9E9, 9E9, 9E9]];
	VAR jointtarget CDP_4529 := [[11.02, 35.4, 6.5, 0, 48.1, -85.27], [9E9, 9E9, 9E9, 9E9, 9E9, 9E9]];
	VAR jointtarget CDP_4530 := [[11.04, 35.41, 6.5, 0, 48.1, -85.91], [9E9, 9E9, 9E9, 9E9, 9E9, 9E9]];
	VAR jointtarget CDP_4531 := [[11.06, 35.41, 6.5, 0, 48.1, -86.56], [9E9, 9E9, 9E9, 9E9, 9E9, 9E9]];
	VAR jointtarget CDP_4532 := [[11.07, 35.41, 6.5, 0, 48.1, -87.2], [9E9, 9E9, 9E9, 9E9, 9E9, 9E9]];
	VAR jointtarget CDP_4533 := [[11.09, 35.41, 6.49, 0, 48.1, -87.85], [9E9, 9E9, 9E9, 9E9, 9E9, 9E9]];
	VAR jointtarget CDP_4534 := [[11.11, 35.41, 6.49, 0, 48.1, -88.49], [9E9, 9E9, 9E9, 9E9, 9E9, 9E9]];
	VAR jointtarget CDP_4535 := [[11.13, 35.41, 6.49, 0, 48.1, -89.14], [9E9, 9E9, 9E9, 9E9, 9E9, 9E9]];
	VAR jointtarget CDP_4536 := [[11.14, 35.41, 6.49, 0, 48.1, -89.78], [9E9, 9E9, 9E9, 9E9, 9E9, 9E9]];
	VAR jointtarget CDP_4537 := [[11.16, 35.41, 6.49, 0, 48.1, -90.43], [9E9, 9E9, 9E9, 9E9, 9E9, 9E9]];
	VAR jointtarget CDP_4538 := [[11.18, 35.41, 6.49, 0, 48.1, -91.07], [9E9, 9E9, 9E9, 9E9, 9E9, 9E9]];
	VAR jointtarget CDP_4539 := [[11.19, 35.41, 6.49, 0, 48.1, -91.72], [9E9, 9E9, 9E9, 9E9, 9E9, 9E9]];
	VAR jointtarget CDP_4540 := [[11.26, 35.4, 6.5, 0, 48.1, -91.98], [9E9, 9E9, 9E9, 9E9, 9E9, 9E9]];
	VAR jointtarget CDP_4541 := [[11.33, 35.4, 6.5, 0, 48.09, -91.91], [9E9, 9E9, 9E9, 9E9, 9E9, 9E9]];
	VAR jointtarget CDP_4542 := [[11.4, 35.4, 6.51, 0, 48.09, -91.84], [9E9, 9E9, 9E9, 9E9, 9E9, 9E9]];
	VAR jointtarget CDP_4543 := [[11.47, 35.4, 6.51, 0, 48.09, -91.78], [9E9, 9E9, 9E9, 9E9, 9E9, 9E9]];
	VAR jointtarget CDP_4544 := [[11.53, 35.4, 6.51, 0, 48.09, -91.71], [9E9, 9E9, 9E9, 9E9, 9E9, 9E9]];
	VAR jointtarget CDP_4545 := [[11.6, 35.39, 6.52, 0, 48.09, -91.64], [9E9, 9E9, 9E9, 9E9, 9E9, 9E9]];
	VAR jointtarget CDP_4546 := [[11.67, 35.39, 6.52, 0, 48.09, -91.57], [9E9, 9E9, 9E9, 9E9, 9E9, 9E9]];
	VAR jointtarget CDP_4547 := [[11.74, 35.39, 6.53, 0, 48.09, -91.5], [9E9, 9E9, 9E9, 9E9, 9E9, 9E9]];
	VAR jointtarget CDP_4548 := [[11.81, 35.39, 6.53, 0, 48.08, -91.44], [9E9, 9E9, 9E9, 9E9, 9E9, 9E9]];
	VAR jointtarget CDP_4549 := [[11.87, 35.39, 6.53, 0, 48.08, -91.37], [9E9, 9E9, 9E9, 9E9, 9E9, 9E9]];
	VAR jointtarget CDP_4550 := [[11.94, 35.38, 6.53, 0, 48.08, -91.3], [9E9, 9E9, 9E9, 9E9, 9E9, 9E9]];
	VAR jointtarget CDP_4551 := [[12.01, 35.38, 6.54, 0, 48.08, -91.23], [9E9, 9E9, 9E9, 9E9, 9E9, 9E9]];
	VAR jointtarget CDP_4552 := [[12.08, 35.38, 6.54, 0, 48.08, -91.16], [9E9, 9E9, 9E9, 9E9, 9E9, 9E9]];
	VAR jointtarget CDP_4553 := [[12.15, 35.38, 6.54, 0, 48.08, -91.09], [9E9, 9E9, 9E9, 9E9, 9E9, 9E9]];
	VAR jointtarget CDP_4554 := [[12.21, 35.38, 6.54, 0, 48.08, -91.03], [9E9, 9E9, 9E9, 9E9, 9E9, 9E9]];
	VAR jointtarget CDP_4555 := [[12.28, 35.38, 6.55, 0, 48.08, -90.96], [9E9, 9E9, 9E9, 9E9, 9E9, 9E9]];
	VAR jointtarget CDP_4556 := [[12.35, 35.38, 6.55, 0, 48.08, -90.89], [9E9, 9E9, 9E9, 9E9, 9E9, 9E9]];
	VAR jointtarget CDP_4557 := [[12.42, 35.37, 6.55, 0, 48.07, -90.82], [9E9, 9E9, 9E9, 9E9, 9E9, 9E9]];
	VAR jointtarget CDP_4558 := [[12.49, 35.37, 6.55, 0, 48.07, -90.75], [9E9, 9E9, 9E9, 9E9, 9E9, 9E9]];
	VAR jointtarget CDP_4559 := [[12.55, 35.37, 6.55, 0, 48.07, -90.69], [9E9, 9E9, 9E9, 9E9, 9E9, 9E9]];
	VAR jointtarget CDP_4560 := [[12.69, 35.38, 6.53, 0, 48.08, -85.39], [9E9, 9E9, 9E9, 9E9, 9E9, 9E9]];
	VAR jointtarget CDP_4561 := [[12.81, 35.42, 6.47, 0, 48.11, -74.94], [9E9, 9E9, 9E9, 9E9, 9E9, 9E9]];
	VAR jointtarget CDP_4562 := [[12.93, 35.48, 6.37, 0, 48.15, -64.5], [9E9, 9E9, 9E9, 9E9, 9E9, 9E9]];
	VAR jointtarget CDP_4563 := [[13.04, 35.57, 6.22, 0, 48.21, -54.07], [9E9, 9E9, 9E9, 9E9, 9E9, 9E9]];
	VAR jointtarget CDP_4564 := [[13.13, 35.67, 6.05, 0, 48.28, -43.65], [9E9, 9E9, 9E9, 9E9, 9E9, 9E9]];
	VAR jointtarget CDP_4565 := [[13.2, 35.79, 5.84, 0, 48.37, -33.25], [9E9, 9E9, 9E9, 9E9, 9E9, 9E9]];
	VAR jointtarget CDP_4566 := [[13.25, 35.92, 5.62, 0, 48.46, -22.88], [9E9, 9E9, 9E9, 9E9, 9E9, 9E9]];
	VAR jointtarget CDP_4567 := [[13.28, 36.06, 5.38, 0, 48.56, -12.53], [9E9, 9E9, 9E9, 9E9, 9E9, 9E9]];
	VAR jointtarget CDP_4568 := [[13.29, 36.2, 5.14, 0, 48.66, -2.2], [9E9, 9E9, 9E9, 9E9, 9E9, 9E9]];
	VAR jointtarget CDP_4569 := [[13.27, 36.34, 4.89, 0, 48.76, 8.11], [9E9, 9E9, 9E9, 9E9, 9E9, 9E9]];
	VAR jointtarget CDP_4570 := [[13.23, 36.48, 4.66, 0, 48.86, 18.39], [9E9, 9E9, 9E9, 9E9, 9E9, 9E9]];
	VAR jointtarget CDP_4571 := [[13.17, 36.61, 4.44, 0, 48.95, 28.65], [9E9, 9E9, 9E9, 9E9, 9E9, 9E9]];
	VAR jointtarget CDP_4572 := [[13.08, 36.72, 4.25, 0, 49.03, 38.9], [9E9, 9E9, 9E9, 9E9, 9E9, 9E9]];
	VAR jointtarget CDP_4573 := [[12.99, 36.81, 4.09, 0, 49.1, 49.12], [9E9, 9E9, 9E9, 9E9, 9E9, 9E9]];
	VAR jointtarget CDP_4574 := [[12.88, 36.89, 3.96, 0, 49.15, 59.33], [9E9, 9E9, 9E9, 9E9, 9E9, 9E9]];
	VAR jointtarget CDP_4575 := [[12.75, 36.94, 3.87, 0, 49.19, 69.54], [9E9, 9E9, 9E9, 9E9, 9E9, 9E9]];
	VAR jointtarget CDP_4576 := [[12.63, 36.96, 3.83, 0, 49.21, 79.73], [9E9, 9E9, 9E9, 9E9, 9E9, 9E9]];
	VAR jointtarget CDP_4577 := [[12.5, 36.96, 3.83, 0, 49.21, 89.93], [9E9, 9E9, 9E9, 9E9, 9E9, 9E9]];
	VAR jointtarget CDP_4578 := [[12.37, 36.94, 3.87, 0, 49.19, 100.13], [9E9, 9E9, 9E9, 9E9, 9E9, 9E9]];
	VAR jointtarget CDP_4579 := [[12.25, 36.89, 3.96, 0, 49.15, 110.33], [9E9, 9E9, 9E9, 9E9, 9E9, 9E9]];
	VAR jointtarget CDP_4580 := [[12.19, 36.86, 4.02, 0, 49.13, 115.43], [9E9, 9E9, 9E9, 9E9, 9E9, 9E9]];
	VAR jointtarget CDP_4581 := [[12.13, 36.82, 4.07, 0, 49.11, 115.37], [9E9, 9E9, 9E9, 9E9, 9E9, 9E9]];
	VAR jointtarget CDP_4582 := [[12.07, 36.79, 4.12, 0, 49.08, 115.31], [9E9, 9E9, 9E9, 9E9, 9E9, 9E9]];
	VAR jointtarget CDP_4583 := [[12.01, 36.76, 4.18, 0, 49.06, 115.25], [9E9, 9E9, 9E9, 9E9, 9E9, 9E9]];
	VAR jointtarget CDP_4584 := [[11.95, 36.73, 4.23, 0, 49.04, 115.19], [9E9, 9E9, 9E9, 9E9, 9E9, 9E9]];
	VAR jointtarget CDP_4585 := [[11.89, 36.7, 4.29, 0, 49.02, 115.13], [9E9, 9E9, 9E9, 9E9, 9E9, 9E9]];
	VAR jointtarget CDP_4586 := [[11.83, 36.67, 4.34, 0, 48.99, 115.07], [9E9, 9E9, 9E9, 9E9, 9E9, 9E9]];
	VAR jointtarget CDP_4587 := [[11.77, 36.63, 4.4, 0, 48.97, 115.01], [9E9, 9E9, 9E9, 9E9, 9E9, 9E9]];
	VAR jointtarget CDP_4588 := [[11.71, 36.6, 4.45, 0, 48.95, 114.95], [9E9, 9E9, 9E9, 9E9, 9E9, 9E9]];
	VAR jointtarget CDP_4589 := [[11.65, 36.57, 4.5, 0, 48.93, 114.89], [9E9, 9E9, 9E9, 9E9, 9E9, 9E9]];
	VAR jointtarget CDP_4590 := [[11.59, 36.54, 4.56, 0, 48.9, 114.83], [9E9, 9E9, 9E9, 9E9, 9E9, 9E9]];
	VAR jointtarget CDP_4591 := [[11.53, 36.51, 4.61, 0, 48.88, 114.77], [9E9, 9E9, 9E9, 9E9, 9E9, 9E9]];
	VAR jointtarget CDP_4592 := [[11.47, 36.48, 4.66, 0, 48.86, 114.71], [9E9, 9E9, 9E9, 9E9, 9E9, 9E9]];
	VAR jointtarget CDP_4593 := [[11.4, 36.45, 4.72, 0, 48.84, 114.64], [9E9, 9E9, 9E9, 9E9, 9E9, 9E9]];
	VAR jointtarget CDP_4594 := [[11.34, 36.42, 4.77, 0, 48.82, 114.58], [9E9, 9E9, 9E9, 9E9, 9E9, 9E9]];
	VAR jointtarget CDP_4595 := [[11.28, 36.39, 4.82, 0, 48.79, 114.52], [9E9, 9E9, 9E9, 9E9, 9E9, 9E9]];
	VAR jointtarget CDP_4596 := [[11.22, 36.36, 4.87, 0, 48.77, 114.46], [9E9, 9E9, 9E9, 9E9, 9E9, 9E9]];
	VAR jointtarget CDP_4597 := [[11.16, 36.33, 4.93, 0, 48.75, 114.4], [9E9, 9E9, 9E9, 9E9, 9E9, 9E9]];
	VAR jointtarget CDP_4598 := [[11.1, 36.29, 4.98, 0, 48.73, 114.34], [9E9, 9E9, 9E9, 9E9, 9E9, 9E9]];
	VAR jointtarget CDP_4599 := [[11.04, 36.26, 5.03, 0, 48.71, 114.28], [9E9, 9E9, 9E9, 9E9, 9E9, 9E9]];
	VAR jointtarget CDP_4600 := [[11.02, 36.26, 5.04, 0, 48.7, 113.93], [9E9, 9E9, 9E9, 9E9, 9E9, 9E9]];
	VAR jointtarget CDP_4601 := [[11.01, 36.25, 5.05, 0, 48.7, 113.26], [9E9, 9E9, 9E9, 9E9, 9E9, 9E9]];
	VAR jointtarget CDP_4602 := [[10.99, 36.24, 5.07, 0, 48.69, 112.58], [9E9, 9E9, 9E9, 9E9, 9E9, 9E9]];
	VAR jointtarget CDP_4603 := [[10.98, 36.24, 5.08, 0, 48.69, 111.9], [9E9, 9E9, 9E9, 9E9, 9E9, 9E9]];
	VAR jointtarget CDP_4604 := [[10.96, 36.23, 5.09, 0, 48.68, 111.22], [9E9, 9E9, 9E9, 9E9, 9E9, 9E9]];
	VAR jointtarget CDP_4605 := [[10.95, 36.22, 5.1, 0, 48.68, 110.55], [9E9, 9E9, 9E9, 9E9, 9E9, 9E9]];
	VAR jointtarget CDP_4606 := [[10.93, 36.22, 5.11, 0, 48.67, 109.87], [9E9, 9E9, 9E9, 9E9, 9E9, 9E9]];
	VAR jointtarget CDP_4607 := [[10.91, 36.21, 5.12, 0, 48.67, 109.19], [9E9, 9E9, 9E9, 9E9, 9E9, 9E9]];
	VAR jointtarget CDP_4608 := [[10.9, 36.2, 5.13, 0, 48.66, 108.51], [9E9, 9E9, 9E9, 9E9, 9E9, 9E9]];
	VAR jointtarget CDP_4609 := [[10.88, 36.2, 5.14, 0, 48.66, 107.83], [9E9, 9E9, 9E9, 9E9, 9E9, 9E9]];
	VAR jointtarget CDP_4610 := [[10.87, 36.19, 5.15, 0, 48.66, 107.16], [9E9, 9E9, 9E9, 9E9, 9E9, 9E9]];
	VAR jointtarget CDP_4611 := [[10.85, 36.19, 5.16, 0, 48.65, 106.48], [9E9, 9E9, 9E9, 9E9, 9E9, 9E9]];
	VAR jointtarget CDP_4612 := [[10.83, 36.18, 5.17, 0, 48.65, 105.8], [9E9, 9E9, 9E9, 9E9, 9E9, 9E9]];
	VAR jointtarget CDP_4613 := [[10.82, 36.18, 5.18, 0, 48.64, 105.12], [9E9, 9E9, 9E9, 9E9, 9E9, 9E9]];
	VAR jointtarget CDP_4614 := [[10.8, 36.17, 5.18, 0, 48.64, 104.44], [9E9, 9E9, 9E9, 9E9, 9E9, 9E9]];
	VAR jointtarget CDP_4615 := [[10.79, 36.17, 5.19, 0, 48.64, 103.77], [9E9, 9E9, 9E9, 9E9, 9E9, 9E9]];
	VAR jointtarget CDP_4616 := [[10.77, 36.17, 5.2, 0, 48.64, 103.09], [9E9, 9E9, 9E9, 9E9, 9E9, 9E9]];
	VAR jointtarget CDP_4617 := [[10.75, 36.16, 5.21, 0, 48.63, 102.41], [9E9, 9E9, 9E9, 9E9, 9E9, 9E9]];
	VAR jointtarget CDP_4618 := [[10.74, 36.16, 5.21, 0, 48.63, 101.73], [9E9, 9E9, 9E9, 9E9, 9E9, 9E9]];
	VAR jointtarget CDP_4619 := [[10.72, 36.15, 5.22, 0, 48.63, 101.05], [9E9, 9E9, 9E9, 9E9, 9E9, 9E9]];
	VAR jointtarget CDP_4620 := [[9.64, 35.94, 5.58, 0, 48.48, 99.64], [9E9, 9E9, 9E9, 9E9, 9E9, 9E9]];
	VAR jointtarget CDP_4621 := [[8.56, 35.75, 5.9, 0, 48.34, 98.56], [9E9, 9E9, 9E9, 9E9, 9E9, 9E9]];
	VAR jointtarget CDP_4622 := [[7.47, 35.59, 6.19, 0, 48.23, 97.47], [9E9, 9E9, 9E9, 9E9, 9E9, 9E9]];
	VAR jointtarget CDP_4623 := [[6.38, 35.44, 6.43, 0, 48.12, 96.38], [9E9, 9E9, 9E9, 9E9, 9E9, 9E9]];
	VAR jointtarget CDP_4624 := [[5.28, 35.32, 6.64, 0, 48.04, 95.28], [9E9, 9E9, 9E9, 9E9, 9E9, 9E9]];
	VAR jointtarget CDP_4625 := [[4.17, 35.23, 6.8, 0, 47.97, 94.17], [9E9, 9E9, 9E9, 9E9, 9E9, 9E9]];
	VAR jointtarget CDP_4626 := [[3.07, 35.15, 6.93, 0, 47.92, 93.07], [9E9, 9E9, 9E9, 9E9, 9E9, 9E9]];
	VAR jointtarget CDP_4627 := [[1.96, 35.1, 7.02, 0, 47.88, 91.96], [9E9, 9E9, 9E9, 9E9, 9E9, 9E9]];
	VAR jointtarget CDP_4628 := [[0.85, 35.07, 7.07, 0, 47.86, 90.85], [9E9, 9E9, 9E9, 9E9, 9E9, 9E9]];
	VAR jointtarget CDP_4629 := [[-0.26, 35.06, 7.08, 0, 47.86, 89.74], [9E9, 9E9, 9E9, 9E9, 9E9, 9E9]];
	VAR jointtarget CDP_4630 := [[-1.37, 35.08, 7.05, 0, 47.87, 88.63], [9E9, 9E9, 9E9, 9E9, 9E9, 9E9]];
	VAR jointtarget CDP_4631 := [[-2.48, 35.12, 6.98, 0, 47.9, 87.52], [9E9, 9E9, 9E9, 9E9, 9E9, 9E9]];
	VAR jointtarget CDP_4632 := [[-3.59, 35.18, 6.88, 0, 47.94, 86.41], [9E9, 9E9, 9E9, 9E9, 9E9, 9E9]];
	VAR jointtarget CDP_4633 := [[-4.7, 35.27, 6.73, 0, 48, 85.3], [9E9, 9E9, 9E9, 9E9, 9E9, 9E9]];
	VAR jointtarget CDP_4634 := [[-5.8, 35.38, 6.54, 0, 48.08, 84.2], [9E9, 9E9, 9E9, 9E9, 9E9, 9E9]];
	VAR jointtarget CDP_4635 := [[-6.9, 35.51, 6.32, 0, 48.17, 83.1], [9E9, 9E9, 9E9, 9E9, 9E9, 9E9]];
	VAR jointtarget CDP_4636 := [[-7.99, 35.66, 6.06, 0, 48.28, 82.01], [9E9, 9E9, 9E9, 9E9, 9E9, 9E9]];
	VAR jointtarget CDP_4637 := [[-9.08, 35.84, 5.75, 0, 48.4, 80.92], [9E9, 9E9, 9E9, 9E9, 9E9, 9E9]];
	VAR jointtarget CDP_4638 := [[-10.16, 36.04, 5.41, 0, 48.55, 79.84], [9E9, 9E9, 9E9, 9E9, 9E9, 9E9]];
	VAR jointtarget CDP_4639 := [[-11.23, 36.26, 5.03, 0, 48.7, 78.77], [9E9, 9E9, 9E9, 9E9, 9E9, 9E9]];
	VAR jointtarget CDP_4640 := [[-11.28, 36.27, 5.01, 0, 48.71, 79.81], [9E9, 9E9, 9E9, 9E9, 9E9, 9E9]];
	VAR jointtarget CDP_4641 := [[-11.34, 36.28, 5, 0, 48.72, 81.95], [9E9, 9E9, 9E9, 9E9, 9E9, 9E9]];
	VAR jointtarget CDP_4642 := [[-11.39, 36.29, 4.99, 0, 48.72, 84.09], [9E9, 9E9, 9E9, 9E9, 9E9, 9E9]];
	VAR jointtarget CDP_4643 := [[-11.45, 36.29, 4.98, 0, 48.73, 86.23], [9E9, 9E9, 9E9, 9E9, 9E9, 9E9]];
	VAR jointtarget CDP_4644 := [[-11.5, 36.29, 4.98, 0, 48.73, 88.37], [9E9, 9E9, 9E9, 9E9, 9E9, 9E9]];
	VAR jointtarget CDP_4645 := [[-11.56, 36.29, 4.98, 0, 48.73, 90.51], [9E9, 9E9, 9E9, 9E9, 9E9, 9E9]];
	VAR jointtarget CDP_4646 := [[-11.61, 36.29, 4.98, 0, 48.72, 92.65], [9E9, 9E9, 9E9, 9E9, 9E9, 9E9]];
	VAR jointtarget CDP_4647 := [[-11.67, 36.29, 4.99, 0, 48.72, 94.78], [9E9, 9E9, 9E9, 9E9, 9E9, 9E9]];
	VAR jointtarget CDP_4648 := [[-11.72, 36.28, 5.01, 0, 48.72, 96.92], [9E9, 9E9, 9E9, 9E9, 9E9, 9E9]];
	VAR jointtarget CDP_4649 := [[-11.78, 36.27, 5.02, 0, 48.71, 99.06], [9E9, 9E9, 9E9, 9E9, 9E9, 9E9]];
	VAR jointtarget CDP_4650 := [[-11.83, 36.26, 5.04, 0, 48.7, 101.2], [9E9, 9E9, 9E9, 9E9, 9E9, 9E9]];
	VAR jointtarget CDP_4651 := [[-11.89, 36.24, 5.07, 0, 48.69, 103.34], [9E9, 9E9, 9E9, 9E9, 9E9, 9E9]];
	VAR jointtarget CDP_4652 := [[-11.94, 36.23, 5.09, 0, 48.68, 105.48], [9E9, 9E9, 9E9, 9E9, 9E9, 9E9]];
	VAR jointtarget CDP_4653 := [[-11.99, 36.21, 5.13, 0, 48.67, 107.63], [9E9, 9E9, 9E9, 9E9, 9E9, 9E9]];
	VAR jointtarget CDP_4654 := [[-12.04, 36.19, 5.16, 0, 48.65, 109.77], [9E9, 9E9, 9E9, 9E9, 9E9, 9E9]];
	VAR jointtarget CDP_4655 := [[-12.09, 36.16, 5.2, 0, 48.64, 111.91], [9E9, 9E9, 9E9, 9E9, 9E9, 9E9]];
	VAR jointtarget CDP_4656 := [[-12.15, 36.14, 5.24, 0, 48.62, 114.05], [9E9, 9E9, 9E9, 9E9, 9E9, 9E9]];
	VAR jointtarget CDP_4657 := [[-12.19, 36.11, 5.29, 0, 48.6, 116.2], [9E9, 9E9, 9E9, 9E9, 9E9, 9E9]];
	VAR jointtarget CDP_4658 := [[-12.24, 36.08, 5.34, 0, 48.58, 118.34], [9E9, 9E9, 9E9, 9E9, 9E9, 9E9]];
	VAR jointtarget CDP_4659 := [[-12.29, 36.05, 5.39, 0, 48.56, 120.49], [9E9, 9E9, 9E9, 9E9, 9E9, 9E9]];
	VAR jointtarget CDP_4660 := [[-12.32, 36.03, 5.42, 0, 48.54, 121.56], [9E9, 9E9, 9E9, 9E9, 9E9, 9E9]];
	VAR jointtarget CDP_4661 := [[-12.35, 36.02, 5.46, 0, 48.53, 121.53], [9E9, 9E9, 9E9, 9E9, 9E9, 9E9]];
	VAR jointtarget CDP_4662 := [[-12.38, 36, 5.49, 0, 48.52, 121.5], [9E9, 9E9, 9E9, 9E9, 9E9, 9E9]];
	VAR jointtarget CDP_4663 := [[-12.41, 35.98, 5.52, 0, 48.5, 121.47], [9E9, 9E9, 9E9, 9E9, 9E9, 9E9]];
	VAR jointtarget CDP_4664 := [[-12.43, 35.96, 5.55, 0, 48.49, 121.44], [9E9, 9E9, 9E9, 9E9, 9E9, 9E9]];
	VAR jointtarget CDP_4665 := [[-12.46, 35.94, 5.59, 0, 48.47, 121.41], [9E9, 9E9, 9E9, 9E9, 9E9, 9E9]];
	VAR jointtarget CDP_4666 := [[-12.49, 35.92, 5.62, 0, 48.46, 121.39], [9E9, 9E9, 9E9, 9E9, 9E9, 9E9]];
	VAR jointtarget CDP_4667 := [[-12.52, 35.9, 5.65, 0, 48.45, 121.36], [9E9, 9E9, 9E9, 9E9, 9E9, 9E9]];
	VAR jointtarget CDP_4668 := [[-12.55, 35.88, 5.68, 0, 48.43, 121.33], [9E9, 9E9, 9E9, 9E9, 9E9, 9E9]];
	VAR jointtarget CDP_4669 := [[-12.58, 35.86, 5.72, 0, 48.42, 121.3], [9E9, 9E9, 9E9, 9E9, 9E9, 9E9]];
	VAR jointtarget CDP_4670 := [[-12.61, 35.84, 5.75, 0, 48.41, 121.27], [9E9, 9E9, 9E9, 9E9, 9E9, 9E9]];
	VAR jointtarget CDP_4671 := [[-12.63, 35.83, 5.78, 0, 48.39, 121.24], [9E9, 9E9, 9E9, 9E9, 9E9, 9E9]];
	VAR jointtarget CDP_4672 := [[-12.66, 35.81, 5.81, 0, 48.38, 121.21], [9E9, 9E9, 9E9, 9E9, 9E9, 9E9]];
	VAR jointtarget CDP_4673 := [[-12.69, 35.79, 5.85, 0, 48.37, 121.18], [9E9, 9E9, 9E9, 9E9, 9E9, 9E9]];
	VAR jointtarget CDP_4674 := [[-12.72, 35.77, 5.88, 0, 48.35, 121.16], [9E9, 9E9, 9E9, 9E9, 9E9, 9E9]];
	VAR jointtarget CDP_4675 := [[-12.75, 35.75, 5.91, 0, 48.34, 121.13], [9E9, 9E9, 9E9, 9E9, 9E9, 9E9]];
	VAR jointtarget CDP_4676 := [[-12.78, 35.73, 5.94, 0, 48.33, 121.1], [9E9, 9E9, 9E9, 9E9, 9E9, 9E9]];
	VAR jointtarget CDP_4677 := [[-12.81, 35.71, 5.98, 0, 48.31, 121.07], [9E9, 9E9, 9E9, 9E9, 9E9, 9E9]];
	VAR jointtarget CDP_4678 := [[-12.84, 35.69, 6.01, 0, 48.3, 121.04], [9E9, 9E9, 9E9, 9E9, 9E9, 9E9]];
	VAR jointtarget CDP_4679 := [[-12.86, 35.67, 6.04, 0, 48.29, 121.01], [9E9, 9E9, 9E9, 9E9, 9E9, 9E9]];
	VAR jointtarget CDP_4680 := [[-13.02, 35.6, 6.16, 0, 48.23, 114.17], [9E9, 9E9, 9E9, 9E9, 9E9, 9E9]];
	VAR jointtarget CDP_4681 := [[-13.18, 35.57, 6.22, 0, 48.21, 100.62], [9E9, 9E9, 9E9, 9E9, 9E9, 9E9]];
	VAR jointtarget CDP_4682 := [[-13.34, 35.58, 6.21, 0, 48.22, 87.07], [9E9, 9E9, 9E9, 9E9, 9E9, 9E9]];
	VAR jointtarget CDP_4683 := [[-13.5, 35.63, 6.12, 0, 48.25, 73.52], [9E9, 9E9, 9E9, 9E9, 9E9, 9E9]];
	VAR jointtarget CDP_4684 := [[-13.64, 35.72, 5.97, 0, 48.32, 59.99], [9E9, 9E9, 9E9, 9E9, 9E9, 9E9]];
	VAR jointtarget CDP_4685 := [[-13.76, 35.84, 5.76, 0, 48.4, 46.48], [9E9, 9E9, 9E9, 9E9, 9E9, 9E9]];
	VAR jointtarget CDP_4686 := [[-13.85, 35.99, 5.5, 0, 48.51, 33.01], [9E9, 9E9, 9E9, 9E9, 9E9, 9E9]];
	VAR jointtarget CDP_4687 := [[-13.91, 36.16, 5.21, 0, 48.63, 19.56], [9E9, 9E9, 9E9, 9E9, 9E9, 9E9]];
	VAR jointtarget CDP_4688 := [[-13.92, 36.34, 4.91, 0, 48.76, 6.16], [9E9, 9E9, 9E9, 9E9, 9E9, 9E9]];
	VAR jointtarget CDP_4689 := [[-13.9, 36.51, 4.6, 0, 48.88, -7.21], [9E9, 9E9, 9E9, 9E9, 9E9, 9E9]];
	VAR jointtarget CDP_4690 := [[-13.85, 36.68, 4.31, 0, 49.01, -20.54], [9E9, 9E9, 9E9, 9E9, 9E9, 9E9]];
	VAR jointtarget CDP_4691 := [[-13.76, 36.83, 4.06, 0, 49.11, -33.84], [9E9, 9E9, 9E9, 9E9, 9E9, 9E9]];
	VAR jointtarget CDP_4692 := [[-13.64, 36.95, 3.85, 0, 49.2, -47.11], [9E9, 9E9, 9E9, 9E9, 9E9, 9E9]];
	VAR jointtarget CDP_4693 := [[-13.5, 37.04, 3.69, 0, 49.27, -60.35], [9E9, 9E9, 9E9, 9E9, 9E9, 9E9]];
	VAR jointtarget CDP_4694 := [[-13.34, 37.09, 3.6, 0, 49.3, -73.59], [9E9, 9E9, 9E9, 9E9, 9E9, 9E9]];
	VAR jointtarget CDP_4695 := [[-13.18, 37.1, 3.59, 0, 49.31, -86.81], [9E9, 9E9, 9E9, 9E9, 9E9, 9E9]];
	VAR jointtarget CDP_4696 := [[-13.02, 37.07, 3.64, 0, 49.29, -100.04], [9E9, 9E9, 9E9, 9E9, 9E9, 9E9]];
	VAR jointtarget CDP_4697 := [[-12.88, 37, 3.77, 0, 49.23, -113.28], [9E9, 9E9, 9E9, 9E9, 9E9, 9E9]];
	VAR jointtarget CDP_4698 := [[-12.75, 36.89, 3.95, 0, 49.16, -126.54], [9E9, 9E9, 9E9, 9E9, 9E9, 9E9]];
	VAR jointtarget CDP_4699 := [[-12.64, 36.76, 4.19, 0, 49.06, -139.82], [9E9, 9E9, 9E9, 9E9, 9E9, 9E9]];
	VAR jointtarget CDP_4700 := [[-12.62, 36.71, 4.26, 0, 49.03, -146.49], [9E9, 9E9, 9E9, 9E9, 9E9, 9E9]];
	VAR jointtarget CDP_4701 := [[-12.59, 36.67, 4.33, 0, 49, -146.47], [9E9, 9E9, 9E9, 9E9, 9E9, 9E9]];
	VAR jointtarget CDP_4702 := [[-12.57, 36.63, 4.4, 0, 48.97, -146.44], [9E9, 9E9, 9E9, 9E9, 9E9, 9E9]];
	VAR jointtarget CDP_4703 := [[-12.54, 36.59, 4.47, 0, 48.94, -146.42], [9E9, 9E9, 9E9, 9E9, 9E9, 9E9]];
	VAR jointtarget CDP_4704 := [[-12.52, 36.55, 4.54, 0, 48.91, -146.4], [9E9, 9E9, 9E9, 9E9, 9E9, 9E9]];
	VAR jointtarget CDP_4705 := [[-12.49, 36.51, 4.61, 0, 48.88, -146.37], [9E9, 9E9, 9E9, 9E9, 9E9, 9E9]];
	VAR jointtarget CDP_4706 := [[-12.47, 36.47, 4.68, 0, 48.85, -146.35], [9E9, 9E9, 9E9, 9E9, 9E9, 9E9]];
	VAR jointtarget CDP_4707 := [[-12.44, 36.43, 4.75, 0, 48.82, -146.32], [9E9, 9E9, 9E9, 9E9, 9E9, 9E9]];
	VAR jointtarget CDP_4708 := [[-12.42, 36.38, 4.82, 0, 48.79, -146.3], [9E9, 9E9, 9E9, 9E9, 9E9, 9E9]];
	VAR jointtarget CDP_4709 := [[-12.39, 36.34, 4.89, 0, 48.76, -146.27], [9E9, 9E9, 9E9, 9E9, 9E9, 9E9]];
	VAR jointtarget CDP_4710 := [[-12.37, 36.3, 4.97, 0, 48.73, -146.25], [9E9, 9E9, 9E9, 9E9, 9E9, 9E9]];
	VAR jointtarget CDP_4711 := [[-12.34, 36.26, 5.04, 0, 48.7, -146.22], [9E9, 9E9, 9E9, 9E9, 9E9, 9E9]];
	VAR jointtarget CDP_4712 := [[-12.32, 36.22, 5.11, 0, 48.67, -146.2], [9E9, 9E9, 9E9, 9E9, 9E9, 9E9]];
	VAR jointtarget CDP_4713 := [[-12.29, 36.18, 5.18, 0, 48.65, -146.17], [9E9, 9E9, 9E9, 9E9, 9E9, 9E9]];
	VAR jointtarget CDP_4714 := [[-12.27, 36.14, 5.25, 0, 48.62, -146.15], [9E9, 9E9, 9E9, 9E9, 9E9, 9E9]];
	VAR jointtarget CDP_4715 := [[-12.24, 36.1, 5.32, 0, 48.59, -146.12], [9E9, 9E9, 9E9, 9E9, 9E9, 9E9]];
	VAR jointtarget CDP_4716 := [[-12.22, 36.06, 5.39, 0, 48.56, -146.1], [9E9, 9E9, 9E9, 9E9, 9E9, 9E9]];
	VAR jointtarget CDP_4717 := [[-12.19, 36.02, 5.46, 0, 48.53, -146.07], [9E9, 9E9, 9E9, 9E9, 9E9, 9E9]];
	VAR jointtarget CDP_4718 := [[-12.17, 35.97, 5.53, 0, 48.5, -146.05], [9E9, 9E9, 9E9, 9E9, 9E9, 9E9]];
	VAR jointtarget CDP_4719 := [[-12.14, 35.93, 5.6, 0, 48.47, -146.02], [9E9, 9E9, 9E9, 9E9, 9E9, 9E9]];
	VAR jointtarget CDP_4720 := [[-12.14, 35.92, 5.62, 0, 48.46, -145.46], [9E9, 9E9, 9E9, 9E9, 9E9, 9E9]];
	VAR jointtarget CDP_4721 := [[-12.13, 35.91, 5.64, 0, 48.45, -144.35], [9E9, 9E9, 9E9, 9E9, 9E9, 9E9]];
	VAR jointtarget CDP_4722 := [[-12.12, 35.9, 5.66, 0, 48.44, -143.24], [9E9, 9E9, 9E9, 9E9, 9E9, 9E9]];
	VAR jointtarget CDP_4723 := [[-12.11, 35.88, 5.68, 0, 48.44, -142.13], [9E9, 9E9, 9E9, 9E9, 9E9, 9E9]];
	VAR jointtarget CDP_4724 := [[-12.1, 35.87, 5.7, 0, 48.43, -141.01], [9E9, 9E9, 9E9, 9E9, 9E9, 9E9]];
	VAR jointtarget CDP_4725 := [[-12.09, 35.86, 5.72, 0, 48.42, -139.9], [9E9, 9E9, 9E9, 9E9, 9E9, 9E9]];
	VAR jointtarget CDP_4726 := [[-12.08, 35.85, 5.74, 0, 48.41, -138.79], [9E9, 9E9, 9E9, 9E9, 9E9, 9E9]];
	VAR jointtarget CDP_4727 := [[-12.07, 35.84, 5.76, 0, 48.4, -137.68], [9E9, 9E9, 9E9, 9E9, 9E9, 9E9]];
	VAR jointtarget CDP_4728 := [[-12.06, 35.83, 5.78, 0, 48.4, -136.56], [9E9, 9E9, 9E9, 9E9, 9E9, 9E9]];
	VAR jointtarget CDP_4729 := [[-12.05, 35.81, 5.8, 0, 48.39, -135.45], [9E9, 9E9, 9E9, 9E9, 9E9, 9E9]];
	VAR jointtarget CDP_4730 := [[-12.04, 35.8, 5.82, 0, 48.38, -134.34], [9E9, 9E9, 9E9, 9E9, 9E9, 9E9]];
	VAR jointtarget CDP_4731 := [[-12.03, 35.79, 5.83, 0, 48.37, -133.22], [9E9, 9E9, 9E9, 9E9, 9E9, 9E9]];
	VAR jointtarget CDP_4732 := [[-12.02, 35.78, 5.85, 0, 48.37, -132.11], [9E9, 9E9, 9E9, 9E9, 9E9, 9E9]];
	VAR jointtarget CDP_4733 := [[-12.01, 35.77, 5.87, 0, 48.36, -130.99], [9E9, 9E9, 9E9, 9E9, 9E9, 9E9]];
	VAR jointtarget CDP_4734 := [[-12, 35.76, 5.88, 0, 48.35, -129.88], [9E9, 9E9, 9E9, 9E9, 9E9, 9E9]];
	VAR jointtarget CDP_4735 := [[-11.99, 35.75, 5.9, 0, 48.35, -128.76], [9E9, 9E9, 9E9, 9E9, 9E9, 9E9]];
	VAR jointtarget CDP_4736 := [[-11.98, 35.74, 5.92, 0, 48.34, -127.65], [9E9, 9E9, 9E9, 9E9, 9E9, 9E9]];
	VAR jointtarget CDP_4737 := [[-11.97, 35.73, 5.93, 0, 48.34, -126.53], [9E9, 9E9, 9E9, 9E9, 9E9, 9E9]];
	VAR jointtarget CDP_4738 := [[-11.96, 35.72, 5.95, 0, 48.33, -125.42], [9E9, 9E9, 9E9, 9E9, 9E9, 9E9]];
	VAR jointtarget CDP_4739 := [[-11.95, 35.71, 5.96, 0, 48.32, -124.3], [9E9, 9E9, 9E9, 9E9, 9E9, 9E9]];
	VAR jointtarget CDP_4740 := [[-11.94, 35.71, 5.97, 0, 48.32, -123.74], [9E9, 9E9, 9E9, 9E9, 9E9, 9E9]];
	VAR jointtarget CDP_4741 := [[-11.93, 35.7, 5.99, 0, 48.31, -123.73], [9E9, 9E9, 9E9, 9E9, 9E9, 9E9]];
	VAR jointtarget CDP_4742 := [[-11.92, 35.69, 6, 0, 48.31, -123.72], [9E9, 9E9, 9E9, 9E9, 9E9, 9E9]];
	VAR jointtarget CDP_4743 := [[-11.9, 35.68, 6.01, 0, 48.3, -123.71], [9E9, 9E9, 9E9, 9E9, 9E9, 9E9]];
	VAR jointtarget CDP_4744 := [[-11.89, 35.67, 6.03, 0, 48.3, -123.7], [9E9, 9E9, 9E9, 9E9, 9E9, 9E9]];
	VAR jointtarget CDP_4745 := [[-11.88, 35.67, 6.04, 0, 48.3, -123.69], [9E9, 9E9, 9E9, 9E9, 9E9, 9E9]];
	VAR jointtarget CDP_4746 := [[-11.87, 35.66, 6.05, 0, 48.29, -123.68], [9E9, 9E9, 9E9, 9E9, 9E9, 9E9]];
	VAR jointtarget CDP_4747 := [[-11.86, 35.65, 6.06, 0, 48.29, -123.66], [9E9, 9E9, 9E9, 9E9, 9E9, 9E9]];
	VAR jointtarget CDP_4748 := [[-11.85, 35.64, 6.08, 0, 48.28, -123.65], [9E9, 9E9, 9E9, 9E9, 9E9, 9E9]];
	VAR jointtarget CDP_4749 := [[-11.84, 35.64, 6.09, 0, 48.28, -123.64], [9E9, 9E9, 9E9, 9E9, 9E9, 9E9]];
	VAR jointtarget CDP_4750 := [[-11.83, 35.63, 6.1, 0, 48.27, -123.63], [9E9, 9E9, 9E9, 9E9, 9E9, 9E9]];
	VAR jointtarget CDP_4751 := [[-11.82, 35.62, 6.11, 0, 48.27, -123.62], [9E9, 9E9, 9E9, 9E9, 9E9, 9E9]];
	VAR jointtarget CDP_4752 := [[-11.81, 35.61, 6.13, 0, 48.26, -123.61], [9E9, 9E9, 9E9, 9E9, 9E9, 9E9]];
	VAR jointtarget CDP_4753 := [[-11.8, 35.6, 6.14, 0, 48.26, -123.6], [9E9, 9E9, 9E9, 9E9, 9E9, 9E9]];
	VAR jointtarget CDP_4754 := [[-11.79, 35.6, 6.15, 0, 48.25, -123.59], [9E9, 9E9, 9E9, 9E9, 9E9, 9E9]];
	VAR jointtarget CDP_4755 := [[-11.78, 35.59, 6.16, 0, 48.25, -123.58], [9E9, 9E9, 9E9, 9E9, 9E9, 9E9]];
	VAR jointtarget CDP_4756 := [[-11.77, 35.58, 6.18, 0, 48.24, -123.57], [9E9, 9E9, 9E9, 9E9, 9E9, 9E9]];
	VAR jointtarget CDP_4757 := [[-11.76, 35.57, 6.19, 0, 48.24, -123.56], [9E9, 9E9, 9E9, 9E9, 9E9, 9E9]];
	VAR jointtarget CDP_4758 := [[-11.75, 35.56, 6.2, 0, 48.23, -123.55], [9E9, 9E9, 9E9, 9E9, 9E9, 9E9]];
	VAR jointtarget CDP_4759 := [[-11.74, 35.56, 6.22, 0, 48.23, -123.54], [9E9, 9E9, 9E9, 9E9, 9E9, 9E9]];
	VAR jointtarget CDP_4760 := [[-10.65, 35.32, 6.61, 0, 48.06, -100.65], [9E9, 9E9, 9E9, 9E9, 9E9, 9E9]];
	VAR jointtarget CDP_4761 := [[-9.55, 35.11, 6.97, 0, 47.92, -99.55], [9E9, 9E9, 9E9, 9E9, 9E9, 9E9]];
	VAR jointtarget CDP_4762 := [[-8.44, 34.93, 7.29, 0, 47.79, -98.44], [9E9, 9E9, 9E9, 9E9, 9E9, 9E9]];
	VAR jointtarget CDP_4763 := [[-7.33, 34.76, 7.57, 0, 47.67, -97.33], [9E9, 9E9, 9E9, 9E9, 9E9, 9E9]];
	VAR jointtarget CDP_4764 := [[-6.21, 34.62, 7.81, 0, 47.57, -96.21], [9E9, 9E9, 9E9, 9E9, 9E9, 9E9]];
	VAR jointtarget CDP_4765 := [[-5.09, 34.51, 8, 0, 47.49, -95.09], [9E9, 9E9, 9E9, 9E9, 9E9, 9E9]];
	VAR jointtarget CDP_4766 := [[-3.96, 34.41, 8.16, 0, 47.43, -93.96], [9E9, 9E9, 9E9, 9E9, 9E9, 9E9]];
	VAR jointtarget CDP_4767 := [[-2.83, 34.34, 8.28, 0, 47.38, -92.83], [9E9, 9E9, 9E9, 9E9, 9E9, 9E9]];
	VAR jointtarget CDP_4768 := [[-1.7, 34.29, 8.36, 0, 47.34, -91.7], [9E9, 9E9, 9E9, 9E9, 9E9, 9E9]];
	VAR jointtarget CDP_4769 := [[-0.56, 34.27, 8.4, 0, 47.33, -90.56], [9E9, 9E9, 9E9, 9E9, 9E9, 9E9]];
	VAR jointtarget CDP_4770 := [[0.57, 34.27, 8.4, 0, 47.33, -89.43], [9E9, 9E9, 9E9, 9E9, 9E9, 9E9]];
	VAR jointtarget CDP_4771 := [[1.7, 34.29, 8.36, 0, 47.34, -88.3], [9E9, 9E9, 9E9, 9E9, 9E9, 9E9]];
	VAR jointtarget CDP_4772 := [[2.84, 34.34, 8.28, 0, 47.38, -87.16], [9E9, 9E9, 9E9, 9E9, 9E9, 9E9]];
	VAR jointtarget CDP_4773 := [[3.97, 34.41, 8.16, 0, 47.43, -86.03], [9E9, 9E9, 9E9, 9E9, 9E9, 9E9]];
	VAR jointtarget CDP_4774 := [[5.09, 34.51, 8, 0, 47.49, -84.91], [9E9, 9E9, 9E9, 9E9, 9E9, 9E9]];
	VAR jointtarget CDP_4775 := [[6.22, 34.62, 7.8, 0, 47.57, -83.78], [9E9, 9E9, 9E9, 9E9, 9E9, 9E9]];
	VAR jointtarget CDP_4776 := [[7.34, 34.76, 7.56, 0, 47.67, -82.66], [9E9, 9E9, 9E9, 9E9, 9E9, 9E9]];
	VAR jointtarget CDP_4777 := [[8.45, 34.93, 7.29, 0, 47.79, -81.55], [9E9, 9E9, 9E9, 9E9, 9E9, 9E9]];
	VAR jointtarget CDP_4778 := [[9.56, 35.12, 6.97, 0, 47.92, -80.44], [9E9, 9E9, 9E9, 9E9, 9E9, 9E9]];
	VAR jointtarget CDP_4779 := [[10.65, 35.33, 6.61, 0, 48.06, -79.35], [9E9, 9E9, 9E9, 9E9, 9E9, 9E9]];
	VAR jointtarget CDP_4780 := [[10.71, 35.34, 6.59, 0, 48.07, -78.19], [9E9, 9E9, 9E9, 9E9, 9E9, 9E9]];
	VAR jointtarget CDP_4781 := [[10.76, 35.35, 6.56, 0, 48.08, -75.95], [9E9, 9E9, 9E9, 9E9, 9E9, 9E9]];
	VAR jointtarget CDP_4782 := [[10.82, 35.37, 6.54, 0, 48.1, -73.7], [9E9, 9E9, 9E9, 9E9, 9E9, 9E9]];
	VAR jointtarget CDP_4783 := [[10.87, 35.39, 6.5, 0, 48.11, -71.45], [9E9, 9E9, 9E9, 9E9, 9E9, 9E9]];
	VAR jointtarget CDP_4784 := [[10.92, 35.41, 6.47, 0, 48.12, -69.2], [9E9, 9E9, 9E9, 9E9, 9E9, 9E9]];
	VAR jointtarget CDP_4785 := [[10.97, 35.43, 6.43, 0, 48.14, -66.96], [9E9, 9E9, 9E9, 9E9, 9E9, 9E9]];
	VAR jointtarget CDP_4786 := [[11.03, 35.46, 6.38, 0, 48.16, -64.72], [9E9, 9E9, 9E9, 9E9, 9E9, 9E9]];
	VAR jointtarget CDP_4787 := [[11.07, 35.49, 6.33, 0, 48.18, -62.47], [9E9, 9E9, 9E9, 9E9, 9E9, 9E9]];
	VAR jointtarget CDP_4788 := [[11.12, 35.52, 6.28, 0, 48.2, -60.23], [9E9, 9E9, 9E9, 9E9, 9E9, 9E9]];
	VAR jointtarget CDP_4789 := [[11.17, 35.55, 6.23, 0, 48.22, -57.99], [9E9, 9E9, 9E9, 9E9, 9E9, 9E9]];
	VAR jointtarget CDP_4790 := [[11.22, 35.58, 6.17, 0, 48.25, -55.75], [9E9, 9E9, 9E9, 9E9, 9E9, 9E9]];
	VAR jointtarget CDP_4791 := [[11.26, 35.62, 6.11, 0, 48.27, -53.51], [9E9, 9E9, 9E9, 9E9, 9E9, 9E9]];
	VAR jointtarget CDP_4792 := [[11.3, 35.66, 6.05, 0, 48.3, -51.27], [9E9, 9E9, 9E9, 9E9, 9E9, 9E9]];
	VAR jointtarget CDP_4793 := [[11.35, 35.7, 5.98, 0, 48.33, -49.04], [9E9, 9E9, 9E9, 9E9, 9E9, 9E9]];
	VAR jointtarget CDP_4794 := [[11.39, 35.74, 5.91, 0, 48.36, -46.8], [9E9, 9E9, 9E9, 9E9, 9E9, 9E9]];
	VAR jointtarget CDP_4795 := [[11.43, 35.78, 5.83, 0, 48.39, -44.57], [9E9, 9E9, 9E9, 9E9, 9E9, 9E9]];
	VAR jointtarget CDP_4796 := [[11.46, 35.82, 5.76, 0, 48.42, -42.34], [9E9, 9E9, 9E9, 9E9, 9E9, 9E9]];
	VAR jointtarget CDP_4797 := [[11.5, 35.87, 5.68, 0, 48.45, -40.11], [9E9, 9E9, 9E9, 9E9, 9E9, 9E9]];
	VAR jointtarget CDP_4798 := [[11.53, 35.92, 5.6, 0, 48.48, -37.88], [9E9, 9E9, 9E9, 9E9, 9E9, 9E9]];
	VAR jointtarget CDP_4799 := [[11.57, 35.97, 5.51, 0, 48.52, -35.65], [9E9, 9E9, 9E9, 9E9, 9E9, 9E9]];
	VAR jointtarget CDP_4800 := [[11.59, 36, 5.46, 0, 48.54, -34.54], [9E9, 9E9, 9E9, 9E9, 9E9, 9E9]];
	VAR jointtarget CDP_4801 := [[11.6, 36.03, 5.41, 0, 48.56, -34.52], [9E9, 9E9, 9E9, 9E9, 9E9, 9E9]];
	VAR jointtarget CDP_4802 := [[11.62, 36.06, 5.36, 0, 48.58, -34.5], [9E9, 9E9, 9E9, 9E9, 9E9, 9E9]];
	VAR jointtarget CDP_4803 := [[11.64, 36.09, 5.31, 0, 48.61, -34.48], [9E9, 9E9, 9E9, 9E9, 9E9, 9E9]];
	VAR jointtarget CDP_4804 := [[11.66, 36.12, 5.25, 0, 48.63, -34.46], [9E9, 9E9, 9E9, 9E9, 9E9, 9E9]];
	VAR jointtarget CDP_4805 := [[11.68, 36.15, 5.2, 0, 48.65, -34.44], [9E9, 9E9, 9E9, 9E9, 9E9, 9E9]];
	VAR jointtarget CDP_4806 := [[11.7, 36.18, 5.15, 0, 48.67, -34.42], [9E9, 9E9, 9E9, 9E9, 9E9, 9E9]];
	VAR jointtarget CDP_4807 := [[11.72, 36.21, 5.1, 0, 48.69, -34.41], [9E9, 9E9, 9E9, 9E9, 9E9, 9E9]];
	VAR jointtarget CDP_4808 := [[11.74, 36.24, 5.05, 0, 48.71, -34.39], [9E9, 9E9, 9E9, 9E9, 9E9, 9E9]];
	VAR jointtarget CDP_4809 := [[11.76, 36.27, 5, 0, 48.73, -34.37], [9E9, 9E9, 9E9, 9E9, 9E9, 9E9]];
	VAR jointtarget CDP_4810 := [[11.77, 36.3, 4.94, 0, 48.76, -34.35], [9E9, 9E9, 9E9, 9E9, 9E9, 9E9]];
	VAR jointtarget CDP_4811 := [[11.79, 36.33, 4.89, 0, 48.78, -34.33], [9E9, 9E9, 9E9, 9E9, 9E9, 9E9]];
	VAR jointtarget CDP_4812 := [[11.81, 36.36, 4.84, 0, 48.8, -34.31], [9E9, 9E9, 9E9, 9E9, 9E9, 9E9]];
	VAR jointtarget CDP_4813 := [[11.83, 36.39, 4.79, 0, 48.82, -34.29], [9E9, 9E9, 9E9, 9E9, 9E9, 9E9]];
	VAR jointtarget CDP_4814 := [[11.85, 36.42, 4.74, 0, 48.84, -34.27], [9E9, 9E9, 9E9, 9E9, 9E9, 9E9]];
	VAR jointtarget CDP_4815 := [[11.87, 36.45, 4.68, 0, 48.86, -34.26], [9E9, 9E9, 9E9, 9E9, 9E9, 9E9]];
	VAR jointtarget CDP_4816 := [[11.89, 36.48, 4.63, 0, 48.89, -34.24], [9E9, 9E9, 9E9, 9E9, 9E9, 9E9]];
	VAR jointtarget CDP_4817 := [[11.91, 36.51, 4.58, 0, 48.91, -34.22], [9E9, 9E9, 9E9, 9E9, 9E9, 9E9]];
	VAR jointtarget CDP_4818 := [[11.92, 36.54, 4.53, 0, 48.93, -34.2], [9E9, 9E9, 9E9, 9E9, 9E9, 9E9]];
	VAR jointtarget CDP_4819 := [[11.94, 36.57, 4.48, 0, 48.95, -34.18], [9E9, 9E9, 9E9, 9E9, 9E9, 9E9]];
	VAR jointtarget CDP_4820 := [[12.05, 36.71, 4.24, 0, 49.05, -40.77], [9E9, 9E9, 9E9, 9E9, 9E9, 9E9]];
	VAR jointtarget CDP_4821 := [[12.18, 36.81, 4.06, 0, 49.13, -54.03], [9E9, 9E9, 9E9, 9E9, 9E9, 9E9]];
	VAR jointtarget CDP_4822 := [[12.33, 36.88, 3.94, 0, 49.18, -67.26], [9E9, 9E9, 9E9, 9E9, 9E9, 9E9]];
	VAR jointtarget CDP_4823 := [[12.49, 36.91, 3.89, 0, 49.2, -80.49], [9E9, 9E9, 9E9, 9E9, 9E9, 9E9]];
	VAR jointtarget CDP_4824 := [[12.65, 36.9, 3.91, 0, 49.19, -93.72], [9E9, 9E9, 9E9, 9E9, 9E9, 9E9]];
	VAR jointtarget CDP_4825 := [[12.8, 36.85, 4, 0, 49.15, -106.95], [9E9, 9E9, 9E9, 9E9, 9E9, 9E9]];
	VAR jointtarget CDP_4826 := [[12.94, 36.76, 4.16, 0, 49.08, -120.2], [9E9, 9E9, 9E9, 9E9, 9E9, 9E9]];
	VAR jointtarget CDP_4827 := [[13.06, 36.63, 4.37, 0, 49, -133.47], [9E9, 9E9, 9E9, 9E9, 9E9, 9E9]];
	VAR jointtarget CDP_4828 := [[13.15, 36.48, 4.63, 0, 48.89, -146.77], [9E9, 9E9, 9E9, 9E9, 9E9, 9E9]];
	VAR jointtarget CDP_4829 := [[13.2, 36.31, 4.92, 0, 48.77, -160.1], [9E9, 9E9, 9E9, 9E9, 9E9, 9E9]];
	VAR jointtarget CDP_4830 := [[13.22, 36.14, 5.22, 0, 48.64, -173.47], [9E9, 9E9, 9E9, 9E9, 9E9, 9E9]];
	VAR jointtarget CDP_4831 := [[13.2, 35.96, 5.53, 0, 48.51, -186.88], [9E9, 9E9, 9E9, 9E9, 9E9, 9E9]];
	VAR jointtarget CDP_4832 := [[13.15, 35.79, 5.81, 0, 48.39, -200.32], [9E9, 9E9, 9E9, 9E9, 9E9, 9E9]];
	VAR jointtarget CDP_4833 := [[13.06, 35.64, 6.07, 0, 48.29, -213.8], [9E9, 9E9, 9E9, 9E9, 9E9, 9E9]];
	VAR jointtarget CDP_4834 := [[12.93, 35.52, 6.27, 0, 48.2, -227.31], [9E9, 9E9, 9E9, 9E9, 9E9, 9E9]];
	VAR jointtarget CDP_4835 := [[12.79, 35.43, 6.42, 0, 48.14, -240.84], [9E9, 9E9, 9E9, 9E9, 9E9, 9E9]];
	VAR jointtarget CDP_4836 := [[12.63, 35.39, 6.51, 0, 48.11, -254.39], [9E9, 9E9, 9E9, 9E9, 9E9, 9E9]];
	VAR jointtarget CDP_4837 := [[12.47, 35.38, 6.52, 0, 48.1, -267.94], [9E9, 9E9, 9E9, 9E9, 9E9, 9E9]];
	VAR jointtarget CDP_4838 := [[12.3, 35.42, 6.46, 0, 48.13, -281.49], [9E9, 9E9, 9E9, 9E9, 9E9, 9E9]];
	VAR jointtarget CDP_4839 := [[12.15, 35.49, 6.33, 0, 48.18, -295.03], [9E9, 9E9, 9E9, 9E9, 9E9, 9E9]];
	VAR jointtarget CDP_4840 := [[12.13, 35.51, 6.3, 0, 48.19, -301.75], [9E9, 9E9, 9E9, 9E9, 9E9, 9E9]];
	VAR jointtarget CDP_4841 := [[12.1, 35.53, 6.26, 0, 48.21, -301.78], [9E9, 9E9, 9E9, 9E9, 9E9, 9E9]];
	VAR jointtarget CDP_4842 := [[12.07, 35.55, 6.23, 0, 48.22, -301.81], [9E9, 9E9, 9E9, 9E9, 9E9, 9E9]];
	VAR jointtarget CDP_4843 := [[12.04, 35.57, 6.2, 0, 48.24, -301.84], [9E9, 9E9, 9E9, 9E9, 9E9, 9E9]];
	VAR jointtarget CDP_4844 := [[12.01, 35.59, 6.16, 0, 48.25, -301.87], [9E9, 9E9, 9E9, 9E9, 9E9, 9E9]];
	VAR jointtarget CDP_4845 := [[11.98, 35.61, 6.13, 0, 48.26, -301.89], [9E9, 9E9, 9E9, 9E9, 9E9, 9E9]];
	VAR jointtarget CDP_4846 := [[11.95, 35.62, 6.1, 0, 48.28, -301.92], [9E9, 9E9, 9E9, 9E9, 9E9, 9E9]];
	VAR jointtarget CDP_4847 := [[11.92, 35.64, 6.07, 0, 48.29, -301.95], [9E9, 9E9, 9E9, 9E9, 9E9, 9E9]];
	VAR jointtarget CDP_4848 := [[11.9, 35.66, 6.03, 0, 48.3, -301.98], [9E9, 9E9, 9E9, 9E9, 9E9, 9E9]];
	VAR jointtarget CDP_4849 := [[11.87, 35.68, 6, 0, 48.32, -302.01], [9E9, 9E9, 9E9, 9E9, 9E9, 9E9]];
	VAR jointtarget CDP_4850 := [[11.84, 35.7, 5.97, 0, 48.33, -302.04], [9E9, 9E9, 9E9, 9E9, 9E9, 9E9]];
	VAR jointtarget CDP_4851 := [[11.81, 35.72, 5.93, 0, 48.34, -302.07], [9E9, 9E9, 9E9, 9E9, 9E9, 9E9]];
	VAR jointtarget CDP_4852 := [[11.78, 35.74, 5.9, 0, 48.36, -302.09], [9E9, 9E9, 9E9, 9E9, 9E9, 9E9]];
	VAR jointtarget CDP_4853 := [[11.75, 35.76, 5.87, 0, 48.37, -302.12], [9E9, 9E9, 9E9, 9E9, 9E9, 9E9]];
	VAR jointtarget CDP_4854 := [[11.73, 35.78, 5.83, 0, 48.39, -302.15], [9E9, 9E9, 9E9, 9E9, 9E9, 9E9]];
	VAR jointtarget CDP_4855 := [[11.7, 35.8, 5.8, 0, 48.4, -302.18], [9E9, 9E9, 9E9, 9E9, 9E9, 9E9]];
